    RBT7_BT_CODE_NO : WORD ;
    RBT7_WELD_COUNT : WORD ;
    RBT8_BT_CODE_NO : WORD ;
    RBT8_WELD_COUNT : WORD ;
    RBT9_BT_CODE_NO : WORD ;
    RBT9_WELD_COUNT : WORD ;
    RBT10_BT_CODE_NO : WORD ;
    RBT10_WELD_COUNT : WORD ;
    RBT11_BT_CODE_NO : WORD ;
    RBT11_WELD_COUNT : WORD ;
    RBT12_BT_CODE_NO : WORD ;
    RBT12_WELD_COUNT : WORD ;
    RBT13_BT_CODE_NO : WORD ;
    RBT13_WELD_COUNT : WORD ;
    RBT14_BT_CODE_NO : WORD ;
    RBT14_WELD_COUNT : WORD ;
    RBT15_BT_CODE_NO : WORD ;
    RBT15_WELD_COUNT : WORD ;
    RBT16_BT_CODE_NO : WORD ;
    RBT16_WELD_COUNT : WORD ;
    RBT17_BT_CODE_NO : WORD ;
    RBT17_WELD_COUNT : WORD ;
    RBT18_BT_CODE_NO : WORD ;
    RBT18_WELD_COUNT : WORD ;
    RBT19_BT_CODE_NO : WORD ;
    RBT19_WELD_COUNT : WORD ;
    RBT20_BT_CODE_NO : WORD ;
    RBT20_WELD_COUNT : WORD ;
    RBT21_BT_CODE_NO : WORD ;
    RBT21_WELD_COUNT : WORD ;
    RBT22_BT_CODE_NO : WORD ;
    RBT22_WELD_COUNT : WORD ;
    RBT23_BT_CODE_NO : WORD ;
    RBT23_WELD_COUNT : WORD ;
    RBT24_BT_CODE_NO : WORD ;
    RBT24_WELD_COUNT : WORD ;
    WELD_DETERMINES_RESULT : WORD ;
    WELD_CHECK_SUM : WORD ;
    SPARE1 : WORD ;
   END_STRUCT ;
  END_STRUCT ;
BEGIN
   S702_WELD_BUFF_DATA1.STATION_MAIN := W#16#0;
   S702_WELD_BUFF_DATA1.DISTINCTION_LH_RH := W#16#0;
   S702_WELD_BUFF_DATA1.STAION_NUMBER := W#16#0;
   S702_WELD_BUFF_DATA1.VIN_NUMBER1 := W#16#0;
   S702_WELD_BUFF_DATA1.VIN_NUMBER2 := W#16#0;
   S702_WELD_BUFF_DATA1.VIN_NUMBER3 := W#16#0;
   S702_WELD_BUFF_DATA1.VIN_NUMBER4 := W#16#0;
   S702_WELD_BUFF_DATA1.SEQ_NUMBER1 := W#16#0;
   S702_WELD_BUFF_DATA1.SEQ_NUMBER2 := W#16#0;
   S702_WELD_BUFF_DATA1.RBT1_BT_CODE_NO := W#16#0;
   S702_WELD_BUFF_DATA1.RBT1_WELD_COUNT := W#16#0;
   S702_WELD_BUFF_DATA1.RBT2_BT_CODE_NO := W#16#0;
   S702_WELD_BUFF_DATA1.RBT2_WELD_COUNT := W#16#0;
   S702_WELD_BUFF_DATA1.RBT3_BT_CODE_NO := W#16#0;
   S702_WELD_BUFF_DATA1.RBT3_WELD_COUNT := W#16#0;
   S702_WELD_BUFF_DATA1.RBT4_BT_CODE_NO := W#16#0;
   S702_WELD_BUFF_DATA1.RBT4_WELD_COUNT := W#16#0;
   S702_WELD_BUFF_DATA1.RBT5_BT_CODE_NO := W#16#0;
   S702_WELD_BUFF_DATA1.RBT5_WELD_COUNT := W#16#0;
   S702_WELD_BUFF_DATA1.RBT6_BT_CODE_NO := W#16#0;
   S702_WELD_BUFF_DATA1.RBT6_WELD_COUNT := W#16#0;
   S702_WELD_BUFF_DATA1.RBT7_BT_CODE_NO := W#16#0;
   S702_WELD_BUFF_DATA1.RBT7_WELD_COUNT := W#16#0;
   S702_WELD_BUFF_DATA1.RBT8_BT_CODE_NO := W#16#0;
   S702_WELD_BUFF_DATA1.RBT8_WELD_COUNT := W#16#0;
   S702_WELD_BUFF_DATA1.RBT9_BT_CODE_NO := W#16#0;
   S702_WELD_BUFF_DATA1.RBT9_WELD_COUNT := W#16#0;
   S702_WELD_BUFF_DATA1.RBT10_BT_CODE_NO := W#16#0;
   S702_WELD_BUFF_DATA1.RBT10_WELD_COUNT := W#16#0;
   S702_WELD_BUFF_DATA1.RBT11_BT_CODE_NO := W#16#0;
   S702_WELD_BUFF_DATA1.RBT11_WELD_COUNT := W#16#0;
   S702_WELD_BUFF_DATA1.RBT12_BT_CODE_NO := W#16#0;
   S702_WELD_BUFF_DATA1.RBT12_WELD_COUNT := W#16#0;
   S702_WELD_BUFF_DATA1.RBT13_BT_CODE_NO := W#16#0;
   S702_WELD_BUFF_DATA1.RBT13_WELD_COUNT := W#16#0;
   S702_WELD_BUFF_DATA1.RBT14_BT_CODE_NO := W#16#0;
   S702_WELD_BUFF_DATA1.RBT14_WELD_COUNT := W#16#0;
   S702_WELD_BUFF_DATA1.RBT15_BT_CODE_NO := W#16#0;
   S702_WELD_BUFF_DATA1.RBT15_WELD_COUNT := W#16#0;
   S702_WELD_BUFF_DATA1.RBT16_BT_CODE_NO := W#16#0;
   S702_WELD_BUFF_DATA1.RBT16_WELD_COUNT := W#16#0;
   S702_WELD_BUFF_DATA1.RBT17_BT_CODE_NO := W#16#0;
   S702_WELD_BUFF_DATA1.RBT17_WELD_COUNT := W#16#0;
   S702_WELD_BUFF_DATA1.RBT18_BT_CODE_NO := W#16#0;
   S702_WELD_BUFF_DATA1.RBT18_WELD_COUNT := W#16#0;
   S702_WELD_BUFF_DATA1.RBT19_BT_CODE_NO := W#16#0;
   S702_WELD_BUFF_DATA1.RBT19_WELD_COUNT := W#16#0;
   S702_WELD_BUFF_DATA1.RBT20_BT_CODE_NO := W#16#0;
   S702_WELD_BUFF_DATA1.RBT20_WELD_COUNT := W#16#0;
   S702_WELD_BUFF_DATA1.RBT21_BT_CODE_NO := W#16#0;
   S702_WELD_BUFF_DATA1.RBT21_WELD_COUNT := W#16#0;
   S702_WELD_BUFF_DATA1.RBT22_BT_CODE_NO := W#16#0;
   S702_WELD_BUFF_DATA1.RBT22_WELD_COUNT := W#16#0;
   S702_WELD_BUFF_DATA1.RBT23_BT_CODE_NO := W#16#0;
   S702_WELD_BUFF_DATA1.RBT23_WELD_COUNT := W#16#0;
   S702_WELD_BUFF_DATA1.RBT24_BT_CODE_NO := W#16#0;
   S702_WELD_BUFF_DATA1.RBT24_WELD_COUNT := W#16#0;
   S702_WELD_BUFF_DATA1.WELD_DETERMINES_RESULT := W#16#0;
   S702_WELD_BUFF_DATA1.WELD_CHECK_SUM := W#16#0;
   S702_WELD_BUFF_DATA1.SPARE1 := W#16#0;
   S702_WELD_BUFF_DATA2.STATION_MAIN := W#16#0;
   S702_WELD_BUFF_DATA2.DISTINCTION_LH_RH := W#16#0;
   S702_WELD_BUFF_DATA2.STAION_NUMBER := W#16#0;
   S702_WELD_BUFF_DATA2.VIN_NUMBER1 := W#16#0;
   S702_WELD_BUFF_DATA2.VIN_NUMBER2 := W#16#0;
   S702_WELD_BUFF_DATA2.VIN_NUMBER3 := W#16#0;
   S702_WELD_BUFF_DATA2.VIN_NUMBER4 := W#16#0;
   S702_WELD_BUFF_DATA2.SEQ_NUMBER1 := W#16#0;
   S702_WELD_BUFF_DATA2.SEQ_NUMBER2 := W#16#0;
   S702_WELD_BUFF_DATA2.RBT1_BT_CODE_NO := W#16#0;
   S702_WELD_BUFF_DATA2.RBT1_WELD_COUNT := W#16#0;
   S702_WELD_BUFF_DATA2.RBT2_BT_CODE_NO := W#16#0;
   S702_WELD_BUFF_DATA2.RBT2_WELD_COUNT := W#16#0;
   S702_WELD_BUFF_DATA2.RBT3_BT_CODE_NO := W#16#0;
   S702_WELD_BUFF_DATA2.RBT3_WELD_COUNT := W#16#0;
   S702_WELD_BUFF_DATA2.RBT4_BT_CODE_NO := W#16#0;
   S702_WELD_BUFF_DATA2.RBT4_WELD_COUNT := W#16#0;
   S702_WELD_BUFF_DATA2.RBT5_BT_CODE_NO := W#16#0;
   S702_WELD_BUFF_DATA2.RBT5_WELD_COUNT := W#16#0;
   S702_WELD_BUFF_DATA2.RBT6_BT_CODE_NO := W#16#0;
   S702_WELD_BUFF_DATA2.RBT6_WELD_COUNT := W#16#0;
   S702_WELD_BUFF_DATA2.RBT7_BT_CODE_NO := W#16#0;
   S702_WELD_BUFF_DATA2.RBT7_WELD_COUNT := W#16#0;
   S702_WELD_BUFF_DATA2.RBT8_BT_CODE_NO := W#16#0;
   S702_WELD_BUFF_DATA2.RBT8_WELD_COUNT := W#16#0;
   S702_WELD_BUFF_DATA2.RBT9_BT_CODE_NO := W#16#0;
   S702_WELD_BUFF_DATA2.RBT9_WELD_COUNT := W#16#0;
   S702_WELD_BUFF_DATA2.RBT10_BT_CODE_NO := W#16#0;
   S702_WELD_BUFF_DATA2.RBT10_WELD_COUNT := W#16#0;
   S702_WELD_BUFF_DATA2.RBT11_BT_CODE_NO := W#16#0;
   S702_WELD_BUFF_DATA2.RBT11_WELD_COUNT := W#16#0;
   S702_WELD_BUFF_DATA2.RBT12_BT_CODE_NO := W#16#0;
   S702_WELD_BUFF_DATA2.RBT12_WELD_COUNT := W#16#0;
   S702_WELD_BUFF_DATA2.RBT13_BT_CODE_NO := W#16#0;
   S702_WELD_BUFF_DATA2.RBT13_WELD_COUNT := W#16#0;
   S702_WELD_BUFF_DATA2.RBT14_BT_CODE_NO := W#16#0;
   S702_WELD_BUFF_DATA2.RBT14_WELD_COUNT := W#16#0;
   S702_WELD_BUFF_DATA2.RBT15_BT_CODE_NO := W#16#0;
   S702_WELD_BUFF_DATA2.RBT15_WELD_COUNT := W#16#0;
   S702_WELD_BUFF_DATA2.RBT16_BT_CODE_NO := W#16#0;
   S702_WELD_BUFF_DATA2.RBT16_WELD_COUNT := W#16#0;
   S702_WELD_BUFF_DATA2.RBT17_BT_CODE_NO := W#16#0;
   S702_WELD_BUFF_DATA2.RBT17_WELD_COUNT := W#16#0;
   S702_WELD_BUFF_DATA2.RBT18_BT_CODE_NO := W#16#0;
   S702_WELD_BUFF_DATA2.RBT18_WELD_COUNT := W#16#0;
   S702_WELD_BUFF_DATA2.RBT19_BT_CODE_NO := W#16#0;
   S702_WELD_BUFF_DATA2.RBT19_WELD_COUNT := W#16#0;
   S702_WELD_BUFF_DATA2.RBT20_BT_CODE_NO := W#16#0;
   S702_WELD_BUFF_DATA2.RBT20_WELD_COUNT := W#16#0;
   S702_WELD_BUFF_DATA2.RBT21_BT_CODE_NO := W#16#0;
   S702_WELD_BUFF_DATA2.RBT21_WELD_COUNT := W#16#0;
   S702_WELD_BUFF_DATA2.RBT22_BT_CODE_NO := W#16#0;
   S702_WELD_BUFF_DATA2.RBT22_WELD_COUNT := W#16#0;
   S702_WELD_BUFF_DATA2.RBT23_BT_CODE_NO := W#16#0;
   S702_WELD_BUFF_DATA2.RBT23_WELD_COUNT := W#16#0;
   S702_WELD_BUFF_DATA2.RBT24_BT_CODE_NO := W#16#0;
   S702_WELD_BUFF_DATA2.RBT24_WELD_COUNT := W#16#0;
   S702_WELD_BUFF_DATA2.WELD_DETERMINES_RESULT := W#16#0;
   S702_WELD_BUFF_DATA2.WELD_CHECK_SUM := W#16#0;
   S702_WELD_BUFF_DATA2.SPARE1 := W#16#0;
   S702_WELD_BUFF_DATA3.STATION_MAIN := W#16#0;
   S702_WELD_BUFF_DATA3.DISTINCTION_LH_RH := W#16#0;
   S702_WELD_BUFF_DATA3.STAION_NUMBER := W#16#0;
   S702_WELD_BUFF_DATA3.VIN_NUMBER1 := W#16#0;
   S702_WELD_BUFF_DATA3.VIN_NUMBER2 := W#16#0;
   S702_WELD_BUFF_DATA3.VIN_NUMBER3 := W#16#0;
   S702_WELD_BUFF_DATA3.VIN_NUMBER4 := W#16#0;
   S702_WELD_BUFF_DATA3.SEQ_NUMBER1 := W#16#0;
   S702_WELD_BUFF_DATA3.SEQ_NUMBER2 := W#16#0;
   S702_WELD_BUFF_DATA3.RBT1_BT_CODE_NO := W#16#0;
   S702_WELD_BUFF_DATA3.RBT1_WELD_COUNT := W#16#0;
   S702_WELD_BUFF_DATA3.RBT2_BT_CODE_NO := W#16#0;
   S702_WELD_BUFF_DATA3.RBT2_WELD_COUNT := W#16#0;
   S702_WELD_BUFF_DATA3.RBT3_BT_CODE_NO := W#16#0;
   S702_WELD_BUFF_DATA3.RBT3_WELD_COUNT := W#16#0;
   S702_WELD_BUFF_DATA3.RBT4_BT_CODE_NO := W#16#0;
   S702_WELD_BUFF_DATA3.RBT4_WELD_COUNT := W#16#0;
   S702_WELD_BUFF_DATA3.RBT5_BT_CODE_NO := W#16#0;
   S702_WELD_BUFF_DATA3.RBT5_WELD_COUNT := W#16#0;
   S702_WELD_BUFF_DATA3.RBT6_BT_CODE_NO := W#16#0;
   S702_WELD_BUFF_DATA3.RBT6_WELD_COUNT := W#16#0;
   S702_WELD_BUFF_DATA3.RBT7_BT_CODE_NO := W#16#0;
   S702_WELD_BUFF_DATA3.RBT7_WELD_COUNT := W#16#0;
   S702_WELD_BUFF_DATA3.RBT8_BT_CODE_NO := W#16#0;
   S702_WELD_BUFF_DATA3.RBT8_WELD_COUNT := W#16#0;
   S702_WELD_BUFF_DATA3.RBT9_BT_CODE_NO := W#16#0;
   S702_WELD_BUFF_DATA3.RBT9_WELD_COUNT := W#16#0;
   S702_WELD_BUFF_DATA3.RBT10_BT_CODE_NO := W#16#0;
   S702_WELD_BUFF_DATA3.RBT10_WELD_COUNT := W#16#0;
   S702_WELD_BUFF_DATA3.RBT11_BT_CODE_NO := W#16#0;
   S702_WELD_BUFF_DATA3.RBT11_WELD_COUNT := W#16#0;
   S702_WELD_BUFF_DATA3.RBT12_BT_CODE_NO := W#16#0;
   S702_WELD_BUFF_DATA3.RBT12_WELD_COUNT := W#16#0;
   S702_WELD_BUFF_DATA3.RBT13_BT_CODE_NO := W#16#0;
   S702_WELD_BUFF_DATA3.RBT13_WELD_COUNT := W#16#0;
   S702_WELD_BUFF_DATA3.RBT14_BT_CODE_NO := W#16#0;
   S702_WELD_BUFF_DATA3.RBT14_WELD_COUNT := W#16#0;
   S702_WELD_BUFF_DATA3.RBT15_BT_CODE_NO := W#16#0;
   S702_WELD_BUFF_DATA3.RBT15_WELD_COUNT := W#16#0;
   S702_WELD_BUFF_DATA3.RBT16_BT_CODE_NO := W#16#0;
   S702_WELD_BUFF_DATA3.RBT16_WELD_COUNT := W#16#0;
   S702_WELD_BUFF_DATA3.RBT17_BT_CODE_NO := W#16#0;
   S702_WELD_BUFF_DATA3.RBT17_WELD_COUNT := W#16#0;
   S702_WELD_BUFF_DATA3.RBT18_BT_CODE_NO := W#16#0;
   S702_WELD_BUFF_DATA3.RBT18_WELD_COUNT := W#16#0;
   S702_WELD_BUFF_DATA3.RBT19_BT_CODE_NO := W#16#0;
   S702_WELD_BUFF_DATA3.RBT19_WELD_COUNT := W#16#0;
   S702_WELD_BUFF_DATA3.RBT20_BT_CODE_NO := W#16#0;
   S702_WELD_BUFF_DATA3.RBT20_WELD_COUNT := W#16#0;
   S702_WELD_BUFF_DATA3.RBT21_BT_CODE_NO := W#16#0;
   S702_WELD_BUFF_DATA3.RBT21_WELD_COUNT := W#16#0;
   S702_WELD_BUFF_DATA3.RBT22_BT_CODE_NO := W#16#0;
   S702_WELD_BUFF_DATA3.RBT22_WELD_COUNT := W#16#0;
   S702_WELD_BUFF_DATA3.RBT23_BT_CODE_NO := W#16#0;
   S702_WELD_BUFF_DATA3.RBT23_WELD_COUNT := W#16#0;
   S702_WELD_BUFF_DATA3.RBT24_BT_CODE_NO := W#16#0;
   S702_WELD_BUFF_DATA3.RBT24_WELD_COUNT := W#16#0;
   S702_WELD_BUFF_DATA3.WELD_DETERMINES_RESULT := W#16#0;
   S702_WELD_BUFF_DATA3.WELD_CHECK_SUM := W#16#0;
   S702_WELD_BUFF_DATA3.SPARE1 := W#16#0;
   S702_WELD_BUFF_DATA4.STATION_MAIN := W#16#0;
   S702_WELD_BUFF_DATA4.DISTINCTION_LH_RH := W#16#0;
   S702_WELD_BUFF_DATA4.STAION_NUMBER := W#16#0;
   S702_WELD_BUFF_DATA4.VIN_NUMBER1 := W#16#0;
   S702_WELD_BUFF_DATA4.VIN_NUMBER2 := W#16#0;
   S702_WELD_BUFF_DATA4.VIN_NUMBER3 := W#16#0;
   S702_WELD_BUFF_DATA4.VIN_NUMBER4 := W#16#0;
   S702_WELD_BUFF_DATA4.SEQ_NUMBER1 := W#16#0;
   S702_WELD_BUFF_DATA4.SEQ_NUMBER2 := W#16#0;
   S702_WELD_BUFF_DATA4.RBT1_BT_CODE_NO := W#16#0;
   S702_WELD_BUFF_DATA4.RBT1_WELD_COUNT := W#16#0;
   S702_WELD_BUFF_DATA4.RBT2_BT_CODE_NO := W#16#0;
   S702_WELD_BUFF_DATA4.RBT2_WELD_COUNT := W#16#0;
   S702_WELD_BUFF_DATA4.RBT3_BT_CODE_NO := W#16#0;
   S702_WELD_BUFF_DATA4.RBT3_WELD_COUNT := W#16#0;
   S702_WELD_BUFF_DATA4.RBT4_BT_CODE_NO := W#16#0;
   S702_WELD_BUFF_DATA4.RBT4_WELD_COUNT := W#16#0;
   S702_WELD_BUFF_DATA4.RBT5_BT_CODE_NO := W#16#0;
   S702_WELD_BUFF_DATA4.RBT5_WELD_COUNT := W#16#0;
   S702_WELD_BUFF_DATA4.RBT6_BT_CODE_NO := W#16#0;
   S702_WELD_BUFF_DATA4.RBT6_WELD_COUNT := W#16#0;
   S702_WELD_BUFF_DATA4.RBT7_BT_CODE_NO := W#16#0;
   S702_WELD_BUFF_DATA4.RBT7_WELD_COUNT := W#16#0;
   S702_WELD_BUFF_DATA4.RBT8_BT_CODE_NO := W#16#0;
   S702_WELD_BUFF_DATA4.RBT8_WELD_COUNT := W#16#0;
   S702_WELD_BUFF_DATA4.RBT9_BT_CODE_NO := W#16#0;
   S702_WELD_BUFF_DATA4.RBT9_WELD_COUNT := W#16#0;
   S702_WELD_BUFF_DATA4.RBT10_BT_CODE_NO := W#16#0;
   S702_WELD_BUFF_DATA4.RBT10_WELD_COUNT := W#16#0;
   S702_WELD_BUFF_DATA4.RBT11_BT_CODE_NO := W#16#0;
   S702_WELD_BUFF_DATA4.RBT11_WELD_COUNT := W#16#0;
   S702_WELD_BUFF_DATA4.RBT12_BT_CODE_NO := W#16#0;
   S702_WELD_BUFF_DATA4.RBT12_WELD_COUNT := W#16#0;
   S702_WELD_BUFF_DATA4.RBT13_BT_CODE_NO := W#16#0;
   S702_WELD_BUFF_DATA4.RBT13_WELD_COUNT := W#16#0;
   S702_WELD_BUFF_DATA4.RBT14_BT_CODE_NO := W#16#0;
   S702_WELD_BUFF_DATA4.RBT14_WELD_COUNT := W#16#0;
   S702_WELD_BUFF_DATA4.RBT15_BT_CODE_NO := W#16#0;
   S702_WELD_BUFF_DATA4.RBT15_WELD_COUNT := W#16#0;
   S702_WELD_BUFF_DATA4.RBT16_BT_CODE_NO := W#16#0;
   S702_WELD_BUFF_DATA4.RBT16_WELD_COUNT := W#16#0;
   S702_WELD_BUFF_DATA4.RBT17_BT_CODE_NO := W#16#0;
   S702_WELD_BUFF_DATA4.RBT17_WELD_COUNT := W#16#0;
   S702_WELD_BUFF_DATA4.RBT18_BT_CODE_NO := W#16#0;
   S702_WELD_BUFF_DATA4.RBT18_WELD_COUNT := W#16#0;
   S702_WELD_BUFF_DATA4.RBT19_BT_CODE_NO := W#16#0;
   S702_WELD_BUFF_DATA4.RBT19_WELD_COUNT := W#16#0;
   S702_WELD_BUFF_DATA4.RBT20_BT_CODE_NO := W#16#0;
   S702_WELD_BUFF_DATA4.RBT20_WELD_COUNT := W#16#0;
   S702_WELD_BUFF_DATA4.RBT21_BT_CODE_NO := W#16#0;
   S702_WELD_BUFF_DATA4.RBT21_WELD_COUNT := W#16#0;
   S702_WELD_BUFF_DATA4.RBT22_BT_CODE_NO := W#16#0;
   S702_WELD_BUFF_DATA4.RBT22_WELD_COUNT := W#16#0;
   S702_WELD_BUFF_DATA4.RBT23_BT_CODE_NO := W#16#0;
   S702_WELD_BUFF_DATA4.RBT23_WELD_COUNT := W#16#0;
   S702_WELD_BUFF_DATA4.RBT24_BT_CODE_NO := W#16#0;
   S702_WELD_BUFF_DATA4.RBT24_WELD_COUNT := W#16#0;
   S702_WELD_BUFF_DATA4.WELD_DETERMINES_RESULT := W#16#0;
   S702_WELD_BUFF_DATA4.WELD_CHECK_SUM := W#16#0;
   S702_WELD_BUFF_DATA4.SPARE1 := W#16#0;
   S702_WELD_BUFF_DATA5.STATION_MAIN := W#16#0;
   S702_WELD_BUFF_DATA5.DISTINCTION_LH_RH := W#16#0;
   S702_WELD_BUFF_DATA5.STAION_NUMBER := W#16#0;
   S702_WELD_BUFF_DATA5.VIN_NUMBER1 := W#16#0;
   S702_WELD_BUFF_DATA5.VIN_NUMBER2 := W#16#0;
   S702_WELD_BUFF_DATA5.VIN_NUMBER3 := W#16#0;
   S702_WELD_BUFF_DATA5.VIN_NUMBER4 := W#16#0;
   S702_WELD_BUFF_DATA5.SEQ_NUMBER1 := W#16#0;
   S702_WELD_BUFF_DATA5.SEQ_NUMBER2 := W#16#0;
   S702_WELD_BUFF_DATA5.RBT1_BT_CODE_NO := W#16#0;
   S702_WELD_BUFF_DATA5.RBT1_WELD_COUNT := W#16#0;
   S702_WELD_BUFF_DATA5.RBT2_BT_CODE_NO := W#16#0;
   S702_WELD_BUFF_DATA5.RBT2_WELD_COUNT := W#16#0;
   S702_WELD_BUFF_DATA5.RBT3_BT_CODE_NO := W#16#0;
   S702_WELD_BUFF_DATA5.RBT3_WELD_COUNT := W#16#0;
   S702_WELD_BUFF_DATA5.RBT4_BT_CODE_NO := W#16#0;
   S702_WELD_BUFF_DATA5.RBT4_WELD_COUNT := W#16#0;
   S702_WELD_BUFF_DATA5.RBT5_BT_CODE_NO := W#16#0;
   S702_WELD_BUFF_DATA5.RBT5_WELD_COUNT := W#16#0;
   S702_WELD_BUFF_DATA5.RBT6_BT_CODE_NO := W#16#0;
   S702_WELD_BUFF_DATA5.RBT6_WELD_COUNT := W#16#0;
   S702_WELD_BUFF_DATA5.RBT7_BT_CODE_NO := W#16#0;
   S702_WELD_BUFF_DATA5.RBT7_WELD_COUNT := W#16#0;
   S702_WELD_BUFF_DATA5.RBT8_BT_CODE_NO := W#16#0;
   S702_WELD_BUFF_DATA5.RBT8_WELD_COUNT := W#16#0;
   S702_WELD_BUFF_DATA5.RBT9_BT_CODE_NO := W#16#0;
   S702_WELD_BUFF_DATA5.RBT9_WELD_COUNT := W#16#0;
   S702_WELD_BUFF_DATA5.RBT10_BT_CODE_NO := W#16#0;
   S702_WELD_BUFF_DATA5.RBT10_WELD_COUNT := W#16#0;
   S702_WELD_BUFF_DATA5.RBT11_BT_CODE_NO := W#16#0;
   S702_WELD_BUFF_DATA5.RBT11_WELD_COUNT := W#16#0;
   S702_WELD_BUFF_DATA5.RBT12_BT_CODE_NO := W#16#0;
   S702_WELD_BUFF_DATA5.RBT12_WELD_COUNT := W#16#0;
   S702_WELD_BUFF_DATA5.RBT13_BT_CODE_NO := W#16#0;
   S702_WELD_BUFF_DATA5.RBT13_WELD_COUNT := W#16#0;
   S702_WELD_BUFF_DATA5.RBT14_BT_CODE_NO := W#16#0;
   S702_WELD_BUFF_DATA5.RBT14_WELD_COUNT := W#16#0;
   S702_WELD_BUFF_DATA5.RBT15_BT_CODE_NO := W#16#0;
   S702_WELD_BUFF_DATA5.RBT15_WELD_COUNT := W#16#0;
   S702_WELD_BUFF_DATA5.RBT16_BT_CODE_NO := W#16#0;
   S702_WELD_BUFF_DATA5.RBT16_WELD_COUNT := W#16#0;
   S702_WELD_BUFF_DATA5.RBT17_BT_CODE_NO := W#16#0;
   S702_WELD_BUFF_DATA5.RBT17_WELD_COUNT := W#16#0;
   S702_WELD_BUFF_DATA5.RBT18_BT_CODE_NO := W#16#0;
   S702_WELD_BUFF_DATA5.RBT18_WELD_COUNT := W#16#0;
   S702_WELD_BUFF_DATA5.RBT19_BT_CODE_NO := W#16#0;
   S702_WELD_BUFF_DATA5.RBT19_WELD_COUNT := W#16#0;
   S702_WELD_BUFF_DATA5.RBT20_BT_CODE_NO := W#16#0;
   S702_WELD_BUFF_DATA5.RBT20_WELD_COUNT := W#16#0;
   S702_WELD_BUFF_DATA5.RBT21_BT_CODE_NO := W#16#0;
   S702_WELD_BUFF_DATA5.RBT21_WELD_COUNT := W#16#0;
   S702_WELD_BUFF_DATA5.RBT22_BT_CODE_NO := W#16#0;
   S702_WELD_BUFF_DATA5.RBT22_WELD_COUNT := W#16#0;
   S702_WELD_BUFF_DATA5.RBT23_BT_CODE_NO := W#16#0;
   S702_WELD_BUFF_DATA5.RBT23_WELD_COUNT := W#16#0;
   S702_WELD_BUFF_DATA5.RBT24_BT_CODE_NO := W#16#0;
   S702_WELD_BUFF_DATA5.RBT24_WELD_COUNT := W#16#0;
   S702_WELD_BUFF_DATA5.WELD_DETERMINES_RESULT := W#16#0;
   S702_WELD_BUFF_DATA5.WELD_CHECK_SUM := W#16#0;
   S702_WELD_BUFF_DATA5.SPARE1 := W#16#0;
   S702_WELD_BUFF_DATA6.STATION_MAIN := W#16#0;
   S702_WELD_BUFF_DATA6.DISTINCTION_LH_RH := W#16#0;
   S702_WELD_BUFF_DATA6.STAION_NUMBER := W#16#0;
   S702_WELD_BUFF_DATA6.VIN_NUMBER1 := W#16#0;
   S702_WELD_BUFF_DATA6.VIN_NUMBER2 := W#16#0;
   S702_WELD_BUFF_DATA6.VIN_NUMBER3 := W#16#0;
   S702_WELD_BUFF_DATA6.VIN_NUMBER4 := W#16#0;
   S702_WELD_BUFF_DATA6.SEQ_NUMBER1 := W#16#0;
   S702_WELD_BUFF_DATA6.SEQ_NUMBER2 := W#16#0;
   S702_WELD_BUFF_DATA6.RBT1_BT_CODE_NO := W#16#0;
   S702_WELD_BUFF_DATA6.RBT1_WELD_COUNT := W#16#0;
   S702_WELD_BUFF_DATA6.RBT2_BT_CODE_NO := W#16#0;
   S702_WELD_BUFF_DATA6.RBT2_WELD_COUNT := W#16#0;
   S702_WELD_BUFF_DATA6.RBT3_BT_CODE_NO := W#16#0;
   S702_WELD_BUFF_DATA6.RBT3_WELD_COUNT := W#16#0;
   S702_WELD_BUFF_DATA6.RBT4_BT_CODE_NO := W#16#0;
   S702_WELD_BUFF_DATA6.RBT4_WELD_COUNT := W#16#0;
   S702_WELD_BUFF_DATA6.RBT5_BT_CODE_NO := W#16#0;
   S702_WELD_BUFF_DATA6.RBT5_WELD_COUNT := W#16#0;
   S702_WELD_BUFF_DATA6.RBT6_BT_CODE_NO := W#16#0;
   S702_WELD_BUFF_DATA6.RBT6_WELD_COUNT := W#16#0;
   S702_WELD_BUFF_DATA6.RBT7_BT_CODE_NO := W#16#0;
   S702_WELD_BUFF_DATA6.RBT7_WELD_COUNT := W#16#0;
   S702_WELD_BUFF_DATA6.RBT8_BT_CODE_NO := W#16#0;
   S702_WELD_BUFF_DATA6.RBT8_WELD_COUNT := W#16#0;
   S702_WELD_BUFF_DATA6.RBT9_BT_CODE_NO := W#16#0;
   S702_WELD_BUFF_DATA6.RBT9_WELD_COUNT := W#16#0;
   S702_WELD_BUFF_DATA6.RBT10_BT_CODE_NO := W#16#0;
   S702_WELD_BUFF_DATA6.RBT10_WELD_COUNT := W#16#0;
   S702_WELD_BUFF_DATA6.RBT11_BT_CODE_NO := W#16#0;
   S702_WELD_BUFF_DATA6.RBT11_WELD_COUNT := W#16#0;
   S702_WELD_BUFF_DATA6.RBT12_BT_CODE_NO := W#16#0;
   S702_WELD_BUFF_DATA6.RBT12_WELD_COUNT := W#16#0;
   S702_WELD_BUFF_DATA6.RBT13_BT_CODE_NO := W#16#0;
   S702_WELD_BUFF_DATA6.RBT13_WELD_COUNT := W#16#0;
   S702_WELD_BUFF_DATA6.RBT14_BT_CODE_NO := W#16#0;
   S702_WELD_BUFF_DATA6.RBT14_WELD_COUNT := W#16#0;
   S702_WELD_BUFF_DATA6.RBT15_BT_CODE_NO := W#16#0;
   S702_WELD_BUFF_DATA6.RBT15_WELD_COUNT := W#16#0;
   S702_WELD_BUFF_DATA6.RBT16_BT_CODE_NO := W#16#0;
   S702_WELD_BUFF_DATA6.RBT16_WELD_COUNT := W#16#0;
   S702_WELD_BUFF_DATA6.RBT17_BT_CODE_NO := W#16#0;
   S702_WELD_BUFF_DATA6.RBT17_WELD_COUNT := W#16#0;
   S702_WELD_BUFF_DATA6.RBT18_BT_CODE_NO := W#16#0;
   S702_WELD_BUFF_DATA6.RBT18_WELD_COUNT := W#16#0;
   S702_WELD_BUFF_DATA6.RBT19_BT_CODE_NO := W#16#0;
   S702_WELD_BUFF_DATA6.RBT19_WELD_COUNT := W#16#0;
   S702_WELD_BUFF_DATA6.RBT20_BT_CODE_NO := W#16#0;
   S702_WELD_BUFF_DATA6.RBT20_WELD_COUNT := W#16#0;
   S702_WELD_BUFF_DATA6.RBT21_BT_CODE_NO := W#16#0;
   S702_WELD_BUFF_DATA6.RBT21_WELD_COUNT := W#16#0;
   S702_WELD_BUFF_DATA6.RBT22_BT_CODE_NO := W#16#0;
   S702_WELD_BUFF_DATA6.RBT22_WELD_COUNT := W#16#0;
   S702_WELD_BUFF_DATA6.RBT23_BT_CODE_NO := W#16#0;
   S702_WELD_BUFF_DATA6.RBT23_WELD_COUNT := W#16#0;
   S702_WELD_BUFF_DATA6.RBT24_BT_CODE_NO := W#16#0;
   S702_WELD_BUFF_DATA6.RBT24_WELD_COUNT := W#16#0;
   S702_WELD_BUFF_DATA6.WELD_DETERMINES_RESULT := W#16#0;
   S702_WELD_BUFF_DATA6.WELD_CHECK_SUM := W#16#0;
   S702_WELD_BUFF_DATA6.SPARE1 := W#16#0;
   S702_WELD_BUFF_DATA7.STATION_MAIN := W#16#0;
   S702_WELD_BUFF_DATA7.DISTINCTION_LH_RH := W#16#0;
   S702_WELD_BUFF_DATA7.STAION_NUMBER := W#16#0;
   S702_WELD_BUFF_DATA7.VIN_NUMBER1 := W#16#0;
   S702_WELD_BUFF_DATA7.VIN_NUMBER2 := W#16#0;
   S702_WELD_BUFF_DATA7.VIN_NUMBER3 := W#16#0;
   S702_WELD_BUFF_DATA7.VIN_NUMBER4 := W#16#0;
   S702_WELD_BUFF_DATA7.SEQ_NUMBER1 := W#16#0;
   S702_WELD_BUFF_DATA7.SEQ_NUMBER2 := W#16#0;
   S702_WELD_BUFF_DATA7.RBT1_BT_CODE_NO := W#16#0;
   S702_WELD_BUFF_DATA7.RBT1_WELD_COUNT := W#16#0;
   S702_WELD_BUFF_DATA7.RBT2_BT_CODE_NO := W#16#0;
   S702_WELD_BUFF_DATA7.RBT2_WELD_COUNT := W#16#0;
   S702_WELD_BUFF_DATA7.RBT3_BT_CODE_NO := W#16#0;
   S702_WELD_BUFF_DATA7.RBT3_WELD_COUNT := W#16#0;
   S702_WELD_BUFF_DATA7.RBT4_BT_CODE_NO := W#16#0;
   S702_WELD_BUFF_DATA7.RBT4_WELD_COUNT := W#16#0;
   S702_WELD_BUFF_DATA7.RBT5_BT_CODE_NO := W#16#0;
   S702_WELD_BUFF_DATA7.RBT5_WELD_COUNT := W#16#0;
   S702_WELD_BUFF_DATA7.RBT6_BT_CODE_NO := W#16#0;
   S702_WELD_BUFF_DATA7.RBT6_WELD_COUNT := W#16#0;
   S702_WELD_BUFF_DATA7.RBT7_BT_CODE_NO := W#16#0;
   S702_WELD_BUFF_DATA7.RBT7_WELD_COUNT := W#16#0;
   S702_WELD_BUFF_DATA7.RBT8_BT_CODE_NO := W#16#0;
   S702_WELD_BUFF_DATA7.RBT8_WELD_COUNT := W#16#0;
   S702_WELD_BUFF_DATA7.RBT9_BT_CODE_NO := W#16#0;
   S702_WELD_BUFF_DATA7.RBT9_WELD_COUNT := W#16#0;
   S702_WELD_BUFF_DATA7.RBT10_BT_CODE_NO := W#16#0;
   S702_WELD_BUFF_DATA7.RBT10_WELD_COUNT := W#16#0;
   S702_WELD_BUFF_DATA7.RBT11_BT_CODE_NO := W#16#0;
   S702_WELD_BUFF_DATA7.RBT11_WELD_COUNT := W#16#0;
   S702_WELD_BUFF_DATA7.RBT12_BT_CODE_NO := W#16#0;
   S702_WELD_BUFF_DATA7.RBT12_WELD_COUNT := W#16#0;
   S702_WELD_BUFF_DATA7.RBT13_BT_CODE_NO := W#16#0;
   S702_WELD_BUFF_DATA7.RBT13_WELD_COUNT := W#16#0;
   S702_WELD_BUFF_DATA7.RBT14_BT_CODE_NO := W#16#0;
   S702_WELD_BUFF_DATA7.RBT14_WELD_COUNT := W#16#0;
   S702_WELD_BUFF_DATA7.RBT15_BT_CODE_NO := W#16#0;
   S702_WELD_BUFF_DATA7.RBT15_WELD_COUNT := W#16#0;
   S702_WELD_BUFF_DATA7.RBT16_BT_CODE_NO := W#16#0;
   S702_WELD_BUFF_DATA7.RBT16_WELD_COUNT := W#16#0;
   S702_WELD_BUFF_DATA7.RBT17_BT_CODE_NO := W#16#0;
   S702_WELD_BUFF_DATA7.RBT17_WELD_COUNT := W#16#0;
   S702_WELD_BUFF_DATA7.RBT18_BT_CODE_NO := W#16#0;
   S702_WELD_BUFF_DATA7.RBT18_WELD_COUNT := W#16#0;
   S702_WELD_BUFF_DATA7.RBT19_BT_CODE_NO := W#16#0;
   S702_WELD_BUFF_DATA7.RBT19_WELD_COUNT := W#16#0;
   S702_WELD_BUFF_DATA7.RBT20_BT_CODE_NO := W#16#0;
   S702_WELD_BUFF_DATA7.RBT20_WELD_COUNT := W#16#0;
   S702_WELD_BUFF_DATA7.RBT21_BT_CODE_NO := W#16#0;
   S702_WELD_BUFF_DATA7.RBT21_WELD_COUNT := W#16#0;
   S702_WELD_BUFF_DATA7.RBT22_BT_CODE_NO := W#16#0;
   S702_WELD_BUFF_DATA7.RBT22_WELD_COUNT := W#16#0;
   S702_WELD_BUFF_DATA7.RBT23_BT_CODE_NO := W#16#0;
   S702_WELD_BUFF_DATA7.RBT23_WELD_COUNT := W#16#0;
   S702_WELD_BUFF_DATA7.RBT24_BT_CODE_NO := W#16#0;
   S702_WELD_BUFF_DATA7.RBT24_WELD_COUNT := W#16#0;
   S702_WELD_BUFF_DATA7.WELD_DETERMINES_RESULT := W#16#0;
   S702_WELD_BUFF_DATA7.WELD_CHECK_SUM := W#16#0;
   S702_WELD_BUFF_DATA7.SPARE1 := W#16#0;
   S702_WELD_BUFF_DATA8.STATION_MAIN := W#16#0;
   S702_WELD_BUFF_DATA8.DISTINCTION_LH_RH := W#16#0;
   S702_WELD_BUFF_DATA8.STAION_NUMBER := W#16#0;
   S702_WELD_BUFF_DATA8.VIN_NUMBER1 := W#16#0;
   S702_WELD_BUFF_DATA8.VIN_NUMBER2 := W#16#0;
   S702_WELD_BUFF_DATA8.VIN_NUMBER3 := W#16#0;
   S702_WELD_BUFF_DATA8.VIN_NUMBER4 := W#16#0;
   S702_WELD_BUFF_DATA8.SEQ_NUMBER1 := W#16#0;
   S702_WELD_BUFF_DATA8.SEQ_NUMBER2 := W#16#0;
   S702_WELD_BUFF_DATA8.RBT1_BT_CODE_NO := W#16#0;
   S702_WELD_BUFF_DATA8.RBT1_WELD_COUNT := W#16#0;
   S702_WELD_BUFF_DATA8.RBT2_BT_CODE_NO := W#16#0;
   S702_WELD_BUFF_DATA8.RBT2_WELD_COUNT := W#16#0;
   S702_WELD_BUFF_DATA8.RBT3_BT_CODE_NO := W#16#0;
   S702_WELD_BUFF_DATA8.RBT3_WELD_COUNT := W#16#0;
   S702_WELD_BUFF_DATA8.RBT4_BT_CODE_NO := W#16#0;
   S702_WELD_BUFF_DATA8.RBT4_WELD_COUNT := W#16#0;
   S702_WELD_BUFF_DATA8.RBT5_BT_CODE_NO := W#16#0;
   S702_WELD_BUFF_DATA8.RBT5_WELD_COUNT := W#16#0;
   S702_WELD_BUFF_DATA8.RBT6_BT_CODE_NO := W#16#0;
   S702_WELD_BUFF_DATA8.RBT6_WELD_COUNT := W#16#0;
   S702_WELD_BUFF_DATA8.RBT7_BT_CODE_NO := W#16#0;
   S702_WELD_BUFF_DATA8.RBT7_WELD_COUNT := W#16#0;
   S702_WELD_BUFF_DATA8.RBT8_BT_CODE_NO := W#16#0;
   S702_WELD_BUFF_DATA8.RBT8_WELD_COUNT := W#16#0;
   S702_WELD_BUFF_DATA8.RBT9_BT_CODE_NO := W#16#0;
   S702_WELD_BUFF_DATA8.RBT9_WELD_COUNT := W#16#0;
   S702_WELD_BUFF_DATA8.RBT10_BT_CODE_NO := W#16#0;
   S702_WELD_BUFF_DATA8.RBT10_WELD_COUNT := W#16#0;
   S702_WELD_BUFF_DATA8.RBT11_BT_CODE_NO := W#16#0;
   S702_WELD_BUFF_DATA8.RBT11_WELD_COUNT := W#16#0;
   S702_WELD_BUFF_DATA8.RBT12_BT_CODE_NO := W#16#0;
   S702_WELD_BUFF_DATA8.RBT12_WELD_COUNT := W#16#0;
   S702_WELD_BUFF_DATA8.RBT13_BT_CODE_NO := W#16#0;
   S702_WELD_BUFF_DATA8.RBT13_WELD_COUNT := W#16#0;
   S702_WELD_BUFF_DATA8.RBT14_BT_CODE_NO := W#16#0;
   S702_WELD_BUFF_DATA8.RBT14_WELD_COUNT := W#16#0;
   S702_WELD_BUFF_DATA8.RBT15_BT_CODE_NO := W#16#0;
   S702_WELD_BUFF_DATA8.RBT15_WELD_COUNT := W#16#0;
   S702_WELD_BUFF_DATA8.RBT16_BT_CODE_NO := W#16#0;
   S702_WELD_BUFF_DATA8.RBT16_WELD_COUNT := W#16#0;
   S702_WELD_BUFF_DATA8.RBT17_BT_CODE_NO := W#16#0;
   S702_WELD_BUFF_DATA8.RBT17_WELD_COUNT := W#16#0;
   S702_WELD_BUFF_DATA8.RBT18_BT_CODE_NO := W#16#0;
   S702_WELD_BUFF_DATA8.RBT18_WELD_COUNT := W#16#0;
   S702_WELD_BUFF_DATA8.RBT19_BT_CODE_NO := W#16#0;
   S702_WELD_BUFF_DATA8.RBT19_WELD_COUNT := W#16#0;
   S702_WELD_BUFF_DATA8.RBT20_BT_CODE_NO := W#16#0;
   S702_WELD_BUFF_DATA8.RBT20_WELD_COUNT := W#16#0;
   S702_WELD_BUFF_DATA8.RBT21_BT_CODE_NO := W#16#0;
   S702_WELD_BUFF_DATA8.RBT21_WELD_COUNT := W#16#0;
   S702_WELD_BUFF_DATA8.RBT22_BT_CODE_NO := W#16#0;
   S702_WELD_BUFF_DATA8.RBT22_WELD_COUNT := W#16#0;
   S702_WELD_BUFF_DATA8.RBT23_BT_CODE_NO := W#16#0;
   S702_WELD_BUFF_DATA8.RBT23_WELD_COUNT := W#16#0;
   S702_WELD_BUFF_DATA8.RBT24_BT_CODE_NO := W#16#0;
   S702_WELD_BUFF_DATA8.RBT24_WELD_COUNT := W#16#0;
   S702_WELD_BUFF_DATA8.WELD_DETERMINES_RESULT := W#16#0;
   S702_WELD_BUFF_DATA8.WELD_CHECK_SUM := W#16#0;
   S702_WELD_BUFF_DATA8.SPARE1 := W#16#0;
   S702_WELD_BUFF_DATA9.STATION_MAIN := W#16#0;
   S702_WELD_BUFF_DATA9.DISTINCTION_LH_RH := W#16#0;
   S702_WELD_BUFF_DATA9.STAION_NUMBER := W#16#0;
   S702_WELD_BUFF_DATA9.VIN_NUMBER1 := W#16#0;
   S702_WELD_BUFF_DATA9.VIN_NUMBER2 := W#16#0;
   S702_WELD_BUFF_DATA9.VIN_NUMBER3 := W#16#0;
   S702_WELD_BUFF_DATA9.VIN_NUMBER4 := W#16#0;
   S702_WELD_BUFF_DATA9.SEQ_NUMBER1 := W#16#0;
   S702_WELD_BUFF_DATA9.SEQ_NUMBER2 := W#16#0;
   S702_WELD_BUFF_DATA9.RBT1_BT_CODE_NO := W#16#0;
   S702_WELD_BUFF_DATA9.RBT1_WELD_COUNT := W#16#0;
   S702_WELD_BUFF_DATA9.RBT2_BT_CODE_NO := W#16#0;
   S702_WELD_BUFF_DATA9.RBT2_WELD_COUNT := W#16#0;
   S702_WELD_BUFF_DATA9.RBT3_BT_CODE_NO := W#16#0;
   S702_WELD_BUFF_DATA9.RBT3_WELD_COUNT := W#16#0;
   S702_WELD_BUFF_DATA9.RBT4_BT_CODE_NO := W#16#0;
   S702_WELD_BUFF_DATA9.RBT4_WELD_COUNT := W#16#0;
   S702_WELD_BUFF_DATA9.RBT5_BT_CODE_NO := W#16#0;
   S702_WELD_BUFF_DATA9.RBT5_WELD_COUNT := W#16#0;
   S702_WELD_BUFF_DATA9.RBT6_BT_CODE_NO := W#16#0;
   S702_WELD_BUFF_DATA9.RBT6_WELD_COUNT := W#16#0;
   S702_WELD_BUFF_DATA9.RBT7_BT_CODE_NO := W#16#0;
   S702_WELD_BUFF_DATA9.RBT7_WELD_COUNT := W#16#0;
   S702_WELD_BUFF_DATA9.RBT8_BT_CODE_NO := W#16#0;
   S702_WELD_BUFF_DATA9.RBT8_WELD_COUNT := W#16#0;
   S702_WELD_BUFF_DATA9.RBT9_BT_CODE_NO := W#16#0;
   S702_WELD_BUFF_DATA9.RBT9_WELD_COUNT := W#16#0;
   S702_WELD_BUFF_DATA9.RBT10_BT_CODE_NO := W#16#0;
   S702_WELD_BUFF_DATA9.RBT10_WELD_COUNT := W#16#0;
   S702_WELD_BUFF_DATA9.RBT11_BT_CODE_NO := W#16#0;
   S702_WELD_BUFF_DATA9.RBT11_WELD_COUNT := W#16#0;
   S702_WELD_BUFF_DATA9.RBT12_BT_CODE_NO := W#16#0;
   S702_WELD_BUFF_DATA9.RBT12_WELD_COUNT := W#16#0;
   S702_WELD_BUFF_DATA9.RBT13_BT_CODE_NO := W#16#0;
   S702_WELD_BUFF_DATA9.RBT13_WELD_COUNT := W#16#0;
   S702_WELD_BUFF_DATA9.RBT14_BT_CODE_NO := W#16#0;
   S702_WELD_BUFF_DATA9.RBT14_WELD_COUNT := W#16#0;
   S702_WELD_BUFF_DATA9.RBT15_BT_CODE_NO := W#16#0;
   S702_WELD_BUFF_DATA9.RBT15_WELD_COUNT := W#16#0;
   S702_WELD_BUFF_DATA9.RBT16_BT_CODE_NO := W#16#0;
   S702_WELD_BUFF_DATA9.RBT16_WELD_COUNT := W#16#0;
   S702_WELD_BUFF_DATA9.RBT17_BT_CODE_NO := W#16#0;
   S702_WELD_BUFF_DATA9.RBT17_WELD_COUNT := W#16#0;
   S702_WELD_BUFF_DATA9.RBT18_BT_CODE_NO := W#16#0;
   S702_WELD_BUFF_DATA9.RBT18_WELD_COUNT := W#16#0;
   S702_WELD_BUFF_DATA9.RBT19_BT_CODE_NO := W#16#0;
   S702_WELD_BUFF_DATA9.RBT19_WELD_COUNT := W#16#0;
   S702_WELD_BUFF_DATA9.RBT20_BT_CODE_NO := W#16#0;
   S702_WELD_BUFF_DATA9.RBT20_WELD_COUNT := W#16#0;
   S702_WELD_BUFF_DATA9.RBT21_BT_CODE_NO := W#16#0;
   S702_WELD_BUFF_DATA9.RBT21_WELD_COUNT := W#16#0;
   S702_WELD_BUFF_DATA9.RBT22_BT_CODE_NO := W#16#0;
   S702_WELD_BUFF_DATA9.RBT22_WELD_COUNT := W#16#0;
   S702_WELD_BUFF_DATA9.RBT23_BT_CODE_NO := W#16#0;
   S702_WELD_BUFF_DATA9.RBT23_WELD_COUNT := W#16#0;
   S702_WELD_BUFF_DATA9.RBT24_BT_CODE_NO := W#16#0;
   S702_WELD_BUFF_DATA9.RBT24_WELD_COUNT := W#16#0;
   S702_WELD_BUFF_DATA9.WELD_DETERMINES_RESULT := W#16#0;
   S702_WELD_BUFF_DATA9.WELD_CHECK_SUM := W#16#0;
   S702_WELD_BUFF_DATA9.SPARE1 := W#16#0;
   S702_WELD_BUFF_DATA10.STATION_MAIN := W#16#0;
   S702_WELD_BUFF_DATA10.DISTINCTION_LH_RH := W#16#0;
   S702_WELD_BUFF_DATA10.STAION_NUMBER := W#16#0;
   S702_WELD_BUFF_DATA10.VIN_NUMBER1 := W#16#0;
   S702_WELD_BUFF_DATA10.VIN_NUMBER2 := W#16#0;
   S702_WELD_BUFF_DATA10.VIN_NUMBER3 := W#16#0;
   S702_WELD_BUFF_DATA10.VIN_NUMBER4 := W#16#0;
   S702_WELD_BUFF_DATA10.SEQ_NUMBER1 := W#16#0;
   S702_WELD_BUFF_DATA10.SEQ_NUMBER2 := W#16#0;
   S702_WELD_BUFF_DATA10.RBT1_BT_CODE_NO := W#16#0;
   S702_WELD_BUFF_DATA10.RBT1_WELD_COUNT := W#16#0;
   S702_WELD_BUFF_DATA10.RBT2_BT_CODE_NO := W#16#0;
   S702_WELD_BUFF_DATA10.RBT2_WELD_COUNT := W#16#0;
   S702_WELD_BUFF_DATA10.RBT3_BT_CODE_NO := W#16#0;
   S702_WELD_BUFF_DATA10.RBT3_WELD_COUNT := W#16#0;
   S702_WELD_BUFF_DATA10.RBT4_BT_CODE_NO := W#16#0;
   S702_WELD_BUFF_DATA10.RBT4_WELD_COUNT := W#16#0;
   S702_WELD_BUFF_DATA10.RBT5_BT_CODE_NO := W#16#0;
   S702_WELD_BUFF_DATA10.RBT5_WELD_COUNT := W#16#0;
   S702_WELD_BUFF_DATA10.RBT6_BT_CODE_NO := W#16#0;
   S702_WELD_BUFF_DATA10.RBT6_WELD_COUNT := W#16#0;
   S702_WELD_BUFF_DATA10.RBT7_BT_CODE_NO := W#16#0;
   S702_WELD_BUFF_DATA10.RBT7_WELD_COUNT := W#16#0;
   S702_WELD_BUFF_DATA10.RBT8_BT_CODE_NO := W#16#0;
   S702_WELD_BUFF_DATA10.RBT8_WELD_COUNT := W#16#0;
   S702_WELD_BUFF_DATA10.RBT9_BT_CODE_NO := W#16#0;
   S702_WELD_BUFF_DATA10.RBT9_WELD_COUNT := W#16#0;
   S702_WELD_BUFF_DATA10.RBT10_BT_CODE_NO := W#16#0;
   S702_WELD_BUFF_DATA10.RBT10_WELD_COUNT := W#16#0;
   S702_WELD_BUFF_DATA10.RBT11_BT_CODE_NO := W#16#0;
   S702_WELD_BUFF_DATA10.RBT11_WELD_COUNT := W#16#0;
   S702_WELD_BUFF_DATA10.RBT12_BT_CODE_NO := W#16#0;
   S702_WELD_BUFF_DATA10.RBT12_WELD_COUNT := W#16#0;
   S702_WELD_BUFF_DATA10.RBT13_BT_CODE_NO := W#16#0;
   S702_WELD_BUFF_DATA10.RBT13_WELD_COUNT := W#16#0;
   S702_WELD_BUFF_DATA10.RBT14_BT_CODE_NO := W#16#0;
   S702_WELD_BUFF_DATA10.RBT14_WELD_COUNT := W#16#0;
   S702_WELD_BUFF_DATA10.RBT15_BT_CODE_NO := W#16#0;
   S702_WELD_BUFF_DATA10.RBT15_WELD_COUNT := W#16#0;
   S702_WELD_BUFF_DATA10.RBT16_BT_CODE_NO := W#16#0;
   S702_WELD_BUFF_DATA10.RBT16_WELD_COUNT := W#16#0;
   S702_WELD_BUFF_DATA10.RBT17_BT_CODE_NO := W#16#0;
   S702_WELD_BUFF_DATA10.RBT17_WELD_COUNT := W#16#0;
   S702_WELD_BUFF_DATA10.RBT18_BT_CODE_NO := W#16#0;
   S702_WELD_BUFF_DATA10.RBT18_WELD_COUNT := W#16#0;
   S702_WELD_BUFF_DATA10.RBT19_BT_CODE_NO := W#16#0;
   S702_WELD_BUFF_DATA10.RBT19_WELD_COUNT := W#16#0;
   S702_WELD_BUFF_DATA10.RBT20_BT_CODE_NO := W#16#0;
   S702_WELD_BUFF_DATA10.RBT20_WELD_COUNT := W#16#0;
   S702_WELD_BUFF_DATA10.RBT21_BT_CODE_NO := W#16#0;
   S702_WELD_BUFF_DATA10.RBT21_WELD_COUNT := W#16#0;
   S702_WELD_BUFF_DATA10.RBT22_BT_CODE_NO := W#16#0;
   S702_WELD_BUFF_DATA10.RBT22_WELD_COUNT := W#16#0;
   S702_WELD_BUFF_DATA10.RBT23_BT_CODE_NO := W#16#0;
   S702_WELD_BUFF_DATA10.RBT23_WELD_COUNT := W#16#0;
   S702_WELD_BUFF_DATA10.RBT24_BT_CODE_NO := W#16#0;
   S702_WELD_BUFF_DATA10.RBT24_WELD_COUNT := W#16#0;
   S702_WELD_BUFF_DATA10.WELD_DETERMINES_RESULT := W#16#0;
   S702_WELD_BUFF_DATA10.WELD_CHECK_SUM := W#16#0;
   S702_WELD_BUFF_DATA10.SPARE1 := W#16#0;
   S703_WELD_BUFF_DATA1.STATION_MAIN := W#16#0;
   S703_WELD_BUFF_DATA1.DISTINCTION_LH_RH := W#16#0;
   S703_WELD_BUFF_DATA1.STAION_NUMBER := W#16#0;
   S703_WELD_BUFF_DATA1.VIN_NUMBER1 := W#16#0;
   S703_WELD_BUFF_DATA1.VIN_NUMBER2 := W#16#0;
   S703_WELD_BUFF_DATA1.VIN_NUMBER3 := W#16#0;
   S703_WELD_BUFF_DATA1.VIN_NUMBER4 := W#16#0;
   S703_WELD_BUFF_DATA1.SEQ_NUMBER1 := W#16#0;
   S703_WELD_BUFF_DATA1.SEQ_NUMBER2 := W#16#0;
   S703_WELD_BUFF_DATA1.RBT1_BT_CODE_NO := W#16#0;
   S703_WELD_BUFF_DATA1.RBT1_WELD_COUNT := W#16#0;
   S703_WELD_BUFF_DATA1.RBT2_BT_CODE_NO := W#16#0;
   S703_WELD_BUFF_DATA1.RBT2_WELD_COUNT := W#16#0;
   S703_WELD_BUFF_DATA1.RBT3_BT_CODE_NO := W#16#0;
   S703_WELD_BUFF_DATA1.RBT3_WELD_COUNT := W#16#0;
   S703_WELD_BUFF_DATA1.RBT4_BT_CODE_NO := W#16#0;
   S703_WELD_BUFF_DATA1.RBT4_WELD_COUNT := W#16#0;
   S703_WELD_BUFF_DATA1.RBT5_BT_CODE_NO := W#16#0;
   S703_WELD_BUFF_DATA1.RBT5_WELD_COUNT := W#16#0;
   S703_WELD_BUFF_DATA1.RBT6_BT_CODE_NO := W#16#0;
   S703_WELD_BUFF_DATA1.RBT6_WELD_COUNT := W#16#0;
   S703_WELD_BUFF_DATA1.RBT7_BT_CODE_NO := W#16#0;
   S703_WELD_BUFF_DATA1.RBT7_WELD_COUNT := W#16#0;
   S703_WELD_BUFF_DATA1.RBT8_BT_CODE_NO := W#16#0;
   S703_WELD_BUFF_DATA1.RBT8_WELD_COUNT := W#16#0;
   S703_WELD_BUFF_DATA1.RBT9_BT_CODE_NO := W#16#0;
   S703_WELD_BUFF_DATA1.RBT9_WELD_COUNT := W#16#0;
   S703_WELD_BUFF_DATA1.RBT10_BT_CODE_NO := W#16#0;
   S703_WELD_BUFF_DATA1.RBT10_WELD_COUNT := W#16#0;
   S703_WELD_BUFF_DATA1.RBT11_BT_CODE_NO := W#16#0;
   S703_WELD_BUFF_DATA1.RBT11_WELD_COUNT := W#16#0;
   S703_WELD_BUFF_DATA1.RBT12_BT_CODE_NO := W#16#0;
   S703_WELD_BUFF_DATA1.RBT12_WELD_COUNT := W#16#0;
   S703_WELD_BUFF_DATA1.RBT13_BT_CODE_NO := W#16#0;
   S703_WELD_BUFF_DATA1.RBT13_WELD_COUNT := W#16#0;
   S703_WELD_BUFF_DATA1.RBT14_BT_CODE_NO := W#16#0;
   S703_WELD_BUFF_DATA1.RBT14_WELD_COUNT := W#16#0;
   S703_WELD_BUFF_DATA1.RBT15_BT_CODE_NO := W#16#0;
   S703_WELD_BUFF_DATA1.RBT15_WELD_COUNT := W#16#0;
   S703_WELD_BUFF_DATA1.RBT16_BT_CODE_NO := W#16#0;
   S703_WELD_BUFF_DATA1.RBT16_WELD_COUNT := W#16#0;
   S703_WELD_BUFF_DATA1.RBT17_BT_CODE_NO := W#16#0;
   S703_WELD_BUFF_DATA1.RBT17_WELD_COUNT := W#16#0;
   S703_WELD_BUFF_DATA1.RBT18_BT_CODE_NO := W#16#0;
   S703_WELD_BUFF_DATA1.RBT18_WELD_COUNT := W#16#0;
   S703_WELD_BUFF_DATA1.RBT19_BT_CODE_NO := W#16#0;
   S703_WELD_BUFF_DATA1.RBT19_WELD_COUNT := W#16#0;
   S703_WELD_BUFF_DATA1.RBT20_BT_CODE_NO := W#16#0;
   S703_WELD_BUFF_DATA1.RBT20_WELD_COUNT := W#16#0;
   S703_WELD_BUFF_DATA1.RBT21_BT_CODE_NO := W#16#0;
   S703_WELD_BUFF_DATA1.RBT21_WELD_COUNT := W#16#0;
   S703_WELD_BUFF_DATA1.RBT22_BT_CODE_NO := W#16#0;
   S703_WELD_BUFF_DATA1.RBT22_WELD_COUNT := W#16#0;
   S703_WELD_BUFF_DATA1.RBT23_BT_CODE_NO := W#16#0;
   S703_WELD_BUFF_DATA1.RBT23_WELD_COUNT := W#16#0;
   S703_WELD_BUFF_DATA1.RBT24_BT_CODE_NO := W#16#0;
   S703_WELD_BUFF_DATA1.RBT24_WELD_COUNT := W#16#0;
   S703_WELD_BUFF_DATA1.WELD_DETERMINES_RESULT := W#16#0;
   S703_WELD_BUFF_DATA1.WELD_CHECK_SUM := W#16#0;
   S703_WELD_BUFF_DATA1.SPARE1 := W#16#0;
   S703_WELD_BUFF_DATA2.STATION_MAIN := W#16#0;
   S703_WELD_BUFF_DATA2.DISTINCTION_LH_RH := W#16#0;
   S703_WELD_BUFF_DATA2.STAION_NUMBER := W#16#0;
   S703_WELD_BUFF_DATA2.VIN_NUMBER1 := W#16#0;
   S703_WELD_BUFF_DATA2.VIN_NUMBER2 := W#16#0;
   S703_WELD_BUFF_DATA2.VIN_NUMBER3 := W#16#0;
   S703_WELD_BUFF_DATA2.VIN_NUMBER4 := W#16#0;
   S703_WELD_BUFF_DATA2.SEQ_NUMBER1 := W#16#0;
   S703_WELD_BUFF_DATA2.SEQ_NUMBER2 := W#16#0;
   S703_WELD_BUFF_DATA2.RBT1_BT_CODE_NO := W#16#0;
   S703_WELD_BUFF_DATA2.RBT1_WELD_COUNT := W#16#0;
   S703_WELD_BUFF_DATA2.RBT2_BT_CODE_NO := W#16#0;
   S703_WELD_BUFF_DATA2.RBT2_WELD_COUNT := W#16#0;
   S703_WELD_BUFF_DATA2.RBT3_BT_CODE_NO := W#16#0;
   S703_WELD_BUFF_DATA2.RBT3_WELD_COUNT := W#16#0;
   S703_WELD_BUFF_DATA2.RBT4_BT_CODE_NO := W#16#0;
   S703_WELD_BUFF_DATA2.RBT4_WELD_COUNT := W#16#0;
   S703_WELD_BUFF_DATA2.RBT5_BT_CODE_NO := W#16#0;
   S703_WELD_BUFF_DATA2.RBT5_WELD_COUNT := W#16#0;
   S703_WELD_BUFF_DATA2.RBT6_BT_CODE_NO := W#16#0;
   S703_WELD_BUFF_DATA2.RBT6_WELD_COUNT := W#16#0;
   S703_WELD_BUFF_DATA2.RBT7_BT_CODE_NO := W#16#0;
   S703_WELD_BUFF_DATA2.RBT7_WELD_COUNT := W#16#0;
   S703_WELD_BUFF_DATA2.RBT8_BT_CODE_NO := W#16#0;
   S703_WELD_BUFF_DATA2.RBT8_WELD_COUNT := W#16#0;
   S703_WELD_BUFF_DATA2.RBT9_BT_CODE_NO := W#16#0;
   S703_WELD_BUFF_DATA2.RBT9_WELD_COUNT := W#16#0;
   S703_WELD_BUFF_DATA2.RBT10_BT_CODE_NO := W#16#0;
   S703_WELD_BUFF_DATA2.RBT10_WELD_COUNT := W#16#0;
   S703_WELD_BUFF_DATA2.RBT11_BT_CODE_NO := W#16#0;
   S703_WELD_BUFF_DATA2.RBT11_WELD_COUNT := W#16#0;
   S703_WELD_BUFF_DATA2.RBT12_BT_CODE_NO := W#16#0;
   S703_WELD_BUFF_DATA2.RBT12_WELD_COUNT := W#16#0;
   S703_WELD_BUFF_DATA2.RBT13_BT_CODE_NO := W#16#0;
   S703_WELD_BUFF_DATA2.RBT13_WELD_COUNT := W#16#0;
   S703_WELD_BUFF_DATA2.RBT14_BT_CODE_NO := W#16#0;
   S703_WELD_BUFF_DATA2.RBT14_WELD_COUNT := W#16#0;
   S703_WELD_BUFF_DATA2.RBT15_BT_CODE_NO := W#16#0;
   S703_WELD_BUFF_DATA2.RBT15_WELD_COUNT := W#16#0;
   S703_WELD_BUFF_DATA2.RBT16_BT_CODE_NO := W#16#0;
   S703_WELD_BUFF_DATA2.RBT16_WELD_COUNT := W#16#0;
   S703_WELD_BUFF_DATA2.RBT17_BT_CODE_NO := W#16#0;
   S703_WELD_BUFF_DATA2.RBT17_WELD_COUNT := W#16#0;
   S703_WELD_BUFF_DATA2.RBT18_BT_CODE_NO := W#16#0;
   S703_WELD_BUFF_DATA2.RBT18_WELD_COUNT := W#16#0;
   S703_WELD_BUFF_DATA2.RBT19_BT_CODE_NO := W#16#0;
   S703_WELD_BUFF_DATA2.RBT19_WELD_COUNT := W#16#0;
   S703_WELD_BUFF_DATA2.RBT20_BT_CODE_NO := W#16#0;
   S703_WELD_BUFF_DATA2.RBT20_WELD_COUNT := W#16#0;
   S703_WELD_BUFF_DATA2.RBT21_BT_CODE_NO := W#16#0;
   S703_WELD_BUFF_DATA2.RBT21_WELD_COUNT := W#16#0;
   S703_WELD_BUFF_DATA2.RBT22_BT_CODE_NO := W#16#0;
   S703_WELD_BUFF_DATA2.RBT22_WELD_COUNT := W#16#0;
   S703_WELD_BUFF_DATA2.RBT23_BT_CODE_NO := W#16#0;
   S703_WELD_BUFF_DATA2.RBT23_WELD_COUNT := W#16#0;
   S703_WELD_BUFF_DATA2.RBT24_BT_CODE_NO := W#16#0;
   S703_WELD_BUFF_DATA2.RBT24_WELD_COUNT := W#16#0;
   S703_WELD_BUFF_DATA2.WELD_DETERMINES_RESULT := W#16#0;
   S703_WELD_BUFF_DATA2.WELD_CHECK_SUM := W#16#0;
   S703_WELD_BUFF_DATA2.SPARE1 := W#16#0;
   S703_WELD_BUFF_DATA3.STATION_MAIN := W#16#0;
   S703_WELD_BUFF_DATA3.DISTINCTION_LH_RH := W#16#0;
   S703_WELD_BUFF_DATA3.STAION_NUMBER := W#16#0;
   S703_WELD_BUFF_DATA3.VIN_NUMBER1 := W#16#0;
   S703_WELD_BUFF_DATA3.VIN_NUMBER2 := W#16#0;
   S703_WELD_BUFF_DATA3.VIN_NUMBER3 := W#16#0;
   S703_WELD_BUFF_DATA3.VIN_NUMBER4 := W#16#0;
   S703_WELD_BUFF_DATA3.SEQ_NUMBER1 := W#16#0;
   S703_WELD_BUFF_DATA3.SEQ_NUMBER2 := W#16#0;
   S703_WELD_BUFF_DATA3.RBT1_BT_CODE_NO := W#16#0;
   S703_WELD_BUFF_DATA3.RBT1_WELD_COUNT := W#16#0;
   S703_WELD_BUFF_DATA3.RBT2_BT_CODE_NO := W#16#0;
   S703_WELD_BUFF_DATA3.RBT2_WELD_COUNT := W#16#0;
   S703_WELD_BUFF_DATA3.RBT3_BT_CODE_NO := W#16#0;
   S703_WELD_BUFF_DATA3.RBT3_WELD_COUNT := W#16#0;
   S703_WELD_BUFF_DATA3.RBT4_BT_CODE_NO := W#16#0;
   S703_WELD_BUFF_DATA3.RBT4_WELD_COUNT := W#16#0;
   S703_WELD_BUFF_DATA3.RBT5_BT_CODE_NO := W#16#0;
   S703_WELD_BUFF_DATA3.RBT5_WELD_COUNT := W#16#0;
   S703_WELD_BUFF_DATA3.RBT6_BT_CODE_NO := W#16#0;
   S703_WELD_BUFF_DATA3.RBT6_WELD_COUNT := W#16#0;
   S703_WELD_BUFF_DATA3.RBT7_BT_CODE_NO := W#16#0;
   S703_WELD_BUFF_DATA3.RBT7_WELD_COUNT := W#16#0;
   S703_WELD_BUFF_DATA3.RBT8_BT_CODE_NO := W#16#0;
   S703_WELD_BUFF_DATA3.RBT8_WELD_COUNT := W#16#0;
   S703_WELD_BUFF_DATA3.RBT9_BT_CODE_NO := W#16#0;
   S703_WELD_BUFF_DATA3.RBT9_WELD_COUNT := W#16#0;
   S703_WELD_BUFF_DATA3.RBT10_BT_CODE_NO := W#16#0;
   S703_WELD_BUFF_DATA3.RBT10_WELD_COUNT := W#16#0;
   S703_WELD_BUFF_DATA3.RBT11_BT_CODE_NO := W#16#0;
   S703_WELD_BUFF_DATA3.RBT11_WELD_COUNT := W#16#0;
   S703_WELD_BUFF_DATA3.RBT12_BT_CODE_NO := W#16#0;
   S703_WELD_BUFF_DATA3.RBT12_WELD_COUNT := W#16#0;
   S703_WELD_BUFF_DATA3.RBT13_BT_CODE_NO := W#16#0;
   S703_WELD_BUFF_DATA3.RBT13_WELD_COUNT := W#16#0;
   S703_WELD_BUFF_DATA3.RBT14_BT_CODE_NO := W#16#0;
   S703_WELD_BUFF_DATA3.RBT14_WELD_COUNT := W#16#0;
   S703_WELD_BUFF_DATA3.RBT15_BT_CODE_NO := W#16#0;
   S703_WELD_BUFF_DATA3.RBT15_WELD_COUNT := W#16#0;
   S703_WELD_BUFF_DATA3.RBT16_BT_CODE_NO := W#16#0;
   S703_WELD_BUFF_DATA3.RBT16_WELD_COUNT := W#16#0;
   S703_WELD_BUFF_DATA3.RBT17_BT_CODE_NO := W#16#0;
   S703_WELD_BUFF_DATA3.RBT17_WELD_COUNT := W#16#0;
   S703_WELD_BUFF_DATA3.RBT18_BT_CODE_NO := W#16#0;
   S703_WELD_BUFF_DATA3.RBT18_WELD_COUNT := W#16#0;
   S703_WELD_BUFF_DATA3.RBT19_BT_CODE_NO := W#16#0;
   S703_WELD_BUFF_DATA3.RBT19_WELD_COUNT := W#16#0;
   S703_WELD_BUFF_DATA3.RBT20_BT_CODE_NO := W#16#0;
   S703_WELD_BUFF_DATA3.RBT20_WELD_COUNT := W#16#0;
   S703_WELD_BUFF_DATA3.RBT21_BT_CODE_NO := W#16#0;
   S703_WELD_BUFF_DATA3.RBT21_WELD_COUNT := W#16#0;
   S703_WELD_BUFF_DATA3.RBT22_BT_CODE_NO := W#16#0;
   S703_WELD_BUFF_DATA3.RBT22_WELD_COUNT := W#16#0;
   S703_WELD_BUFF_DATA3.RBT23_BT_CODE_NO := W#16#0;
   S703_WELD_BUFF_DATA3.RBT23_WELD_COUNT := W#16#0;
   S703_WELD_BUFF_DATA3.RBT24_BT_CODE_NO := W#16#0;
   S703_WELD_BUFF_DATA3.RBT24_WELD_COUNT := W#16#0;
   S703_WELD_BUFF_DATA3.WELD_DETERMINES_RESULT := W#16#0;
   S703_WELD_BUFF_DATA3.WELD_CHECK_SUM := W#16#0;
   S703_WELD_BUFF_DATA3.SPARE1 := W#16#0;
   S703_WELD_BUFF_DATA4.STATION_MAIN := W#16#0;
   S703_WELD_BUFF_DATA4.DISTINCTION_LH_RH := W#16#0;
   S703_WELD_BUFF_DATA4.STAION_NUMBER := W#16#0;
   S703_WELD_BUFF_DATA4.VIN_NUMBER1 := W#16#0;
   S703_WELD_BUFF_DATA4.VIN_NUMBER2 := W#16#0;
   S703_WELD_BUFF_DATA4.VIN_NUMBER3 := W#16#0;
   S703_WELD_BUFF_DATA4.VIN_NUMBER4 := W#16#0;
   S703_WELD_BUFF_DATA4.SEQ_NUMBER1 := W#16#0;
   S703_WELD_BUFF_DATA4.SEQ_NUMBER2 := W#16#0;
   S703_WELD_BUFF_DATA4.RBT1_BT_CODE_NO := W#16#0;
   S703_WELD_BUFF_DATA4.RBT1_WELD_COUNT := W#16#0;
   S703_WELD_BUFF_DATA4.RBT2_BT_CODE_NO := W#16#0;
   S703_WELD_BUFF_DATA4.RBT2_WELD_COUNT := W#16#0;
   S703_WELD_BUFF_DATA4.RBT3_BT_CODE_NO := W#16#0;
   S703_WELD_BUFF_DATA4.RBT3_WELD_COUNT := W#16#0;
   S703_WELD_BUFF_DATA4.RBT4_BT_CODE_NO := W#16#0;
   S703_WELD_BUFF_DATA4.RBT4_WELD_COUNT := W#16#0;
   S703_WELD_BUFF_DATA4.RBT5_BT_CODE_NO := W#16#0;
   S703_WELD_BUFF_DATA4.RBT5_WELD_COUNT := W#16#0;
   S703_WELD_BUFF_DATA4.RBT6_BT_CODE_NO := W#16#0;
   S703_WELD_BUFF_DATA4.RBT6_WELD_COUNT := W#16#0;
   S703_WELD_BUFF_DATA4.RBT7_BT_CODE_NO := W#16#0;
   S703_WELD_BUFF_DATA4.RBT7_WELD_COUNT := W#16#0;
   S703_WELD_BUFF_DATA4.RBT8_BT_CODE_NO := W#16#0;
   S703_WELD_BUFF_DATA4.RBT8_WELD_COUNT := W#16#0;
   S703_WELD_BUFF_DATA4.RBT9_BT_CODE_NO := W#16#0;
   S703_WELD_BUFF_DATA4.RBT9_WELD_COUNT := W#16#0;
   S703_WELD_BUFF_DATA4.RBT10_BT_CODE_NO := W#16#0;
   S703_WELD_BUFF_DATA4.RBT10_WELD_COUNT := W#16#0;
   S703_WELD_BUFF_DATA4.RBT11_BT_CODE_NO := W#16#0;
   S703_WELD_BUFF_DATA4.RBT11_WELD_COUNT := W#16#0;
   S703_WELD_BUFF_DATA4.RBT12_BT_CODE_NO := W#16#0;
   S703_WELD_BUFF_DATA4.RBT12_WELD_COUNT := W#16#0;
   S703_WELD_BUFF_DATA4.RBT13_BT_CODE_NO := W#16#0;
   S703_WELD_BUFF_DATA4.RBT13_WELD_COUNT := W#16#0;
   S703_WELD_BUFF_DATA4.RBT14_BT_CODE_NO := W#16#0;
   S703_WELD_BUFF_DATA4.RBT14_WELD_COUNT := W#16#0;
   S703_WELD_BUFF_DATA4.RBT15_BT_CODE_NO := W#16#0;
   S703_WELD_BUFF_DATA4.RBT15_WELD_COUNT := W#16#0;
   S703_WELD_BUFF_DATA4.RBT16_BT_CODE_NO := W#16#0;
   S703_WELD_BUFF_DATA4.RBT16_WELD_COUNT := W#16#0;
   S703_WELD_BUFF_DATA4.RBT17_BT_CODE_NO := W#16#0;
   S703_WELD_BUFF_DATA4.RBT17_WELD_COUNT := W#16#0;
   S703_WELD_BUFF_DATA4.RBT18_BT_CODE_NO := W#16#0;
   S703_WELD_BUFF_DATA4.RBT18_WELD_COUNT := W#16#0;
   S703_WELD_BUFF_DATA4.RBT19_BT_CODE_NO := W#16#0;
   S703_WELD_BUFF_DATA4.RBT19_WELD_COUNT := W#16#0;
   S703_WELD_BUFF_DATA4.RBT20_BT_CODE_NO := W#16#0;
   S703_WELD_BUFF_DATA4.RBT20_WELD_COUNT := W#16#0;
   S703_WELD_BUFF_DATA4.RBT21_BT_CODE_NO := W#16#0;
   S703_WELD_BUFF_DATA4.RBT21_WELD_COUNT := W#16#0;
   S703_WELD_BUFF_DATA4.RBT22_BT_CODE_NO := W#16#0;
   S703_WELD_BUFF_DATA4.RBT22_WELD_COUNT := W#16#0;
   S703_WELD_BUFF_DATA4.RBT23_BT_CODE_NO := W#16#0;
   S703_WELD_BUFF_DATA4.RBT23_WELD_COUNT := W#16#0;
   S703_WELD_BUFF_DATA4.RBT24_BT_CODE_NO := W#16#0;
   S703_WELD_BUFF_DATA4.RBT24_WELD_COUNT := W#16#0;
   S703_WELD_BUFF_DATA4.WELD_DETERMINES_RESULT := W#16#0;
   S703_WELD_BUFF_DATA4.WELD_CHECK_SUM := W#16#0;
   S703_WELD_BUFF_DATA4.SPARE1 := W#16#0;
   S703_WELD_BUFF_DATA5.STATION_MAIN := W#16#0;
   S703_WELD_BUFF_DATA5.DISTINCTION_LH_RH := W#16#0;
   S703_WELD_BUFF_DATA5.STAION_NUMBER := W#16#0;
   S703_WELD_BUFF_DATA5.VIN_NUMBER1 := W#16#0;
   S703_WELD_BUFF_DATA5.VIN_NUMBER2 := W#16#0;
   S703_WELD_BUFF_DATA5.VIN_NUMBER3 := W#16#0;
   S703_WELD_BUFF_DATA5.VIN_NUMBER4 := W#16#0;
   S703_WELD_BUFF_DATA5.SEQ_NUMBER1 := W#16#0;
   S703_WELD_BUFF_DATA5.SEQ_NUMBER2 := W#16#0;
   S703_WELD_BUFF_DATA5.RBT1_BT_CODE_NO := W#16#0;
   S703_WELD_BUFF_DATA5.RBT1_WELD_COUNT := W#16#0;
   S703_WELD_BUFF_DATA5.RBT2_BT_CODE_NO := W#16#0;
   S703_WELD_BUFF_DATA5.RBT2_WELD_COUNT := W#16#0;
   S703_WELD_BUFF_DATA5.RBT3_BT_CODE_NO := W#16#0;
   S703_WELD_BUFF_DATA5.RBT3_WELD_COUNT := W#16#0;
   S703_WELD_BUFF_DATA5.RBT4_BT_CODE_NO := W#16#0;
   S703_WELD_BUFF_DATA5.RBT4_WELD_COUNT := W#16#0;
   S703_WELD_BUFF_DATA5.RBT5_BT_CODE_NO := W#16#0;
   S703_WELD_BUFF_DATA5.RBT5_WELD_COUNT := W#16#0;
   S703_WELD_BUFF_DATA5.RBT6_BT_CODE_NO := W#16#0;
   S703_WELD_BUFF_DATA5.RBT6_WELD_COUNT := W#16#0;
   S703_WELD_BUFF_DATA5.RBT7_BT_CODE_NO := W#16#0;
   S703_WELD_BUFF_DATA5.RBT7_WELD_COUNT := W#16#0;
   S703_WELD_BUFF_DATA5.RBT8_BT_CODE_NO := W#16#0;
   S703_WELD_BUFF_DATA5.RBT8_WELD_COUNT := W#16#0;
   S703_WELD_BUFF_DATA5.RBT9_BT_CODE_NO := W#16#0;
   S703_WELD_BUFF_DATA5.RBT9_WELD_COUNT := W#16#0;
   S703_WELD_BUFF_DATA5.RBT10_BT_CODE_NO := W#16#0;
   S703_WELD_BUFF_DATA5.RBT10_WELD_COUNT := W#16#0;
   S703_WELD_BUFF_DATA5.RBT11_BT_CODE_NO := W#16#0;
   S703_WELD_BUFF_DATA5.RBT11_WELD_COUNT := W#16#0;
   S703_WELD_BUFF_DATA5.RBT12_BT_CODE_NO := W#16#0;
   S703_WELD_BUFF_DATA5.RBT12_WELD_COUNT := W#16#0;
   S703_WELD_BUFF_DATA5.RBT13_BT_CODE_NO := W#16#0;
   S703_WELD_BUFF_DATA5.RBT13_WELD_COUNT := W#16#0;
   S703_WELD_BUFF_DATA5.RBT14_BT_CODE_NO := W#16#0;
   S703_WELD_BUFF_DATA5.RBT14_WELD_COUNT := W#16#0;
   S703_WELD_BUFF_DATA5.RBT15_BT_CODE_NO := W#16#0;
   S703_WELD_BUFF_DATA5.RBT15_WELD_COUNT := W#16#0;
   S703_WELD_BUFF_DATA5.RBT16_BT_CODE_NO := W#16#0;
   S703_WELD_BUFF_DATA5.RBT16_WELD_COUNT := W#16#0;
   S703_WELD_BUFF_DATA5.RBT17_BT_CODE_NO := W#16#0;
   S703_WELD_BUFF_DATA5.RBT17_WELD_COUNT := W#16#0;
   S703_WELD_BUFF_DATA5.RBT18_BT_CODE_NO := W#16#0;
   S703_WELD_BUFF_DATA5.RBT18_WELD_COUNT := W#16#0;
   S703_WELD_BUFF_DATA5.RBT19_BT_CODE_NO := W#16#0;
   S703_WELD_BUFF_DATA5.RBT19_WELD_COUNT := W#16#0;
   S703_WELD_BUFF_DATA5.RBT20_BT_CODE_NO := W#16#0;
   S703_WELD_BUFF_DATA5.RBT20_WELD_COUNT := W#16#0;
   S703_WELD_BUFF_DATA5.RBT21_BT_CODE_NO := W#16#0;
   S703_WELD_BUFF_DATA5.RBT21_WELD_COUNT := W#16#0;
   S703_WELD_BUFF_DATA5.RBT22_BT_CODE_NO := W#16#0;
   S703_WELD_BUFF_DATA5.RBT22_WELD_COUNT := W#16#0;
   S703_WELD_BUFF_DATA5.RBT23_BT_CODE_NO := W#16#0;
   S703_WELD_BUFF_DATA5.RBT23_WELD_COUNT := W#16#0;
   S703_WELD_BUFF_DATA5.RBT24_BT_CODE_NO := W#16#0;
   S703_WELD_BUFF_DATA5.RBT24_WELD_COUNT := W#16#0;
   S703_WELD_BUFF_DATA5.WELD_DETERMINES_RESULT := W#16#0;
   S703_WELD_BUFF_DATA5.WELD_CHECK_SUM := W#16#0;
   S703_WELD_BUFF_DATA5.SPARE1 := W#16#0;
   S703_WELD_BUFF_DATA6.STATION_MAIN := W#16#0;
   S703_WELD_BUFF_DATA6.DISTINCTION_LH_RH := W#16#0;
   S703_WELD_BUFF_DATA6.STAION_NUMBER := W#16#0;
   S703_WELD_BUFF_DATA6.VIN_NUMBER1 := W#16#0;
   S703_WELD_BUFF_DATA6.VIN_NUMBER2 := W#16#0;
   S703_WELD_BUFF_DATA6.VIN_NUMBER3 := W#16#0;
   S703_WELD_BUFF_DATA6.VIN_NUMBER4 := W#16#0;
   S703_WELD_BUFF_DATA6.SEQ_NUMBER1 := W#16#0;
   S703_WELD_BUFF_DATA6.SEQ_NUMBER2 := W#16#0;
   S703_WELD_BUFF_DATA6.RBT1_BT_CODE_NO := W#16#0;
   S703_WELD_BUFF_DATA6.RBT1_WELD_COUNT := W#16#0;
   S703_WELD_BUFF_DATA6.RBT2_BT_CODE_NO := W#16#0;
   S703_WELD_BUFF_DATA6.RBT2_WELD_COUNT := W#16#0;
   S703_WELD_BUFF_DATA6.RBT3_BT_CODE_NO := W#16#0;
   S703_WELD_BUFF_DATA6.RBT3_WELD_COUNT := W#16#0;
   S703_WELD_BUFF_DATA6.RBT4_BT_CODE_NO := W#16#0;
   S703_WELD_BUFF_DATA6.RBT4_WELD_COUNT := W#16#0;
   S703_WELD_BUFF_DATA6.RBT5_BT_CODE_NO := W#16#0;
   S703_WELD_BUFF_DATA6.RBT5_WELD_COUNT := W#16#0;
   S703_WELD_BUFF_DATA6.RBT6_BT_CODE_NO := W#16#0;
   S703_WELD_BUFF_DATA6.RBT6_WELD_COUNT := W#16#0;
   S703_WELD_BUFF_DATA6.RBT7_BT_CODE_NO := W#16#0;
   S703_WELD_BUFF_DATA6.RBT7_WELD_COUNT := W#16#0;
   S703_WELD_BUFF_DATA6.RBT8_BT_CODE_NO := W#16#0;
   S703_WELD_BUFF_DATA6.RBT8_WELD_COUNT := W#16#0;
   S703_WELD_BUFF_DATA6.RBT9_BT_CODE_NO := W#16#0;
   S703_WELD_BUFF_DATA6.RBT9_WELD_COUNT := W#16#0;
   S703_WELD_BUFF_DATA6.RBT10_BT_CODE_NO := W#16#0;
   S703_WELD_BUFF_DATA6.RBT10_WELD_COUNT := W#16#0;
   S703_WELD_BUFF_DATA6.RBT11_BT_CODE_NO := W#16#0;
   S703_WELD_BUFF_DATA6.RBT11_WELD_COUNT := W#16#0;
   S703_WELD_BUFF_DATA6.RBT12_BT_CODE_NO := W#16#0;
   S703_WELD_BUFF_DATA6.RBT12_WELD_COUNT := W#16#0;
   S703_WELD_BUFF_DATA6.RBT13_BT_CODE_NO := W#16#0;
   S703_WELD_BUFF_DATA6.RBT13_WELD_COUNT := W#16#0;
   S703_WELD_BUFF_DATA6.RBT14_BT_CODE_NO := W#16#0;
   S703_WELD_BUFF_DATA6.RBT14_WELD_COUNT := W#16#0;
   S703_WELD_BUFF_DATA6.RBT15_BT_CODE_NO := W#16#0;
   S703_WELD_BUFF_DATA6.RBT15_WELD_COUNT := W#16#0;
   S703_WELD_BUFF_DATA6.RBT16_BT_CODE_NO := W#16#0;
   S703_WELD_BUFF_DATA6.RBT16_WELD_COUNT := W#16#0;
   S703_WELD_BUFF_DATA6.RBT17_BT_CODE_NO := W#16#0;
   S703_WELD_BUFF_DATA6.RBT17_WELD_COUNT := W#16#0;
   S703_WELD_BUFF_DATA6.RBT18_BT_CODE_NO := W#16#0;
   S703_WELD_BUFF_DATA6.RBT18_WELD_COUNT := W#16#0;
   S703_WELD_BUFF_DATA6.RBT19_BT_CODE_NO := W#16#0;
   S703_WELD_BUFF_DATA6.RBT19_WELD_COUNT := W#16#0;
   S703_WELD_BUFF_DATA6.RBT20_BT_CODE_NO := W#16#0;
   S703_WELD_BUFF_DATA6.RBT20_WELD_COUNT := W#16#0;
   S703_WELD_BUFF_DATA6.RBT21_BT_CODE_NO := W#16#0;
   S703_WELD_BUFF_DATA6.RBT21_WELD_COUNT := W#16#0;
   S703_WELD_BUFF_DATA6.RBT22_BT_CODE_NO := W#16#0;
   S703_WELD_BUFF_DATA6.RBT22_WELD_COUNT := W#16#0;
   S703_WELD_BUFF_DATA6.RBT23_BT_CODE_NO := W#16#0;
   S703_WELD_BUFF_DATA6.RBT23_WELD_COUNT := W#16#0;
   S703_WELD_BUFF_DATA6.RBT24_BT_CODE_NO := W#16#0;
   S703_WELD_BUFF_DATA6.RBT24_WELD_COUNT := W#16#0;
   S703_WELD_BUFF_DATA6.WELD_DETERMINES_RESULT := W#16#0;
   S703_WELD_BUFF_DATA6.WELD_CHECK_SUM := W#16#0;
   S703_WELD_BUFF_DATA6.SPARE1 := W#16#0;
   S703_WELD_BUFF_DATA7.STATION_MAIN := W#16#0;
   S703_WELD_BUFF_DATA7.DISTINCTION_LH_RH := W#16#0;
   S703_WELD_BUFF_DATA7.STAION_NUMBER := W#16#0;
   S703_WELD_BUFF_DATA7.VIN_NUMBER1 := W#16#0;
   S703_WELD_BUFF_DATA7.VIN_NUMBER2 := W#16#0;
   S703_WELD_BUFF_DATA7.VIN_NUMBER3 := W#16#0;
   S703_WELD_BUFF_DATA7.VIN_NUMBER4 := W#16#0;
   S703_WELD_BUFF_DATA7.SEQ_NUMBER1 := W#16#0;
   S703_WELD_BUFF_DATA7.SEQ_NUMBER2 := W#16#0;
   S703_WELD_BUFF_DATA7.RBT1_BT_CODE_NO := W#16#0;
   S703_WELD_BUFF_DATA7.RBT1_WELD_COUNT := W#16#0;
   S703_WELD_BUFF_DATA7.RBT2_BT_CODE_NO := W#16#0;
   S703_WELD_BUFF_DATA7.RBT2_WELD_COUNT := W#16#0;
   S703_WELD_BUFF_DATA7.RBT3_BT_CODE_NO := W#16#0;
   S703_WELD_BUFF_DATA7.RBT3_WELD_COUNT := W#16#0;
   S703_WELD_BUFF_DATA7.RBT4_BT_CODE_NO := W#16#0;
   S703_WELD_BUFF_DATA7.RBT4_WELD_COUNT := W#16#0;
   S703_WELD_BUFF_DATA7.RBT5_BT_CODE_NO := W#16#0;
   S703_WELD_BUFF_DATA7.RBT5_WELD_COUNT := W#16#0;
   S703_WELD_BUFF_DATA7.RBT6_BT_CODE_NO := W#16#0;
   S703_WELD_BUFF_DATA7.RBT6_WELD_COUNT := W#16#0;
   S703_WELD_BUFF_DATA7.RBT7_BT_CODE_NO := W#16#0;
   S703_WELD_BUFF_DATA7.RBT7_WELD_COUNT := W#16#0;
   S703_WELD_BUFF_DATA7.RBT8_BT_CODE_NO := W#16#0;
   S703_WELD_BUFF_DATA7.RBT8_WELD_COUNT := W#16#0;
   S703_WELD_BUFF_DATA7.RBT9_BT_CODE_NO := W#16#0;
   S703_WELD_BUFF_DATA7.RBT9_WELD_COUNT := W#16#0;
   S703_WELD_BUFF_DATA7.RBT10_BT_CODE_NO := W#16#0;
   S703_WELD_BUFF_DATA7.RBT10_WELD_COUNT := W#16#0;
   S703_WELD_BUFF_DATA7.RBT11_BT_CODE_NO := W#16#0;
   S703_WELD_BUFF_DATA7.RBT11_WELD_COUNT := W#16#0;
   S703_WELD_BUFF_DATA7.RBT12_BT_CODE_NO := W#16#0;
   S703_WELD_BUFF_DATA7.RBT12_WELD_COUNT := W#16#0;
   S703_WELD_BUFF_DATA7.RBT13_BT_CODE_NO := W#16#0;
   S703_WELD_BUFF_DATA7.RBT13_WELD_COUNT := W#16#0;
   S703_WELD_BUFF_DATA7.RBT14_BT_CODE_NO := W#16#0;
   S703_WELD_BUFF_DATA7.RBT14_WELD_COUNT := W#16#0;
   S703_WELD_BUFF_DATA7.RBT15_BT_CODE_NO := W#16#0;
   S703_WELD_BUFF_DATA7.RBT15_WELD_COUNT := W#16#0;
   S703_WELD_BUFF_DATA7.RBT16_BT_CODE_NO := W#16#0;
   S703_WELD_BUFF_DATA7.RBT16_WELD_COUNT := W#16#0;
   S703_WELD_BUFF_DATA7.RBT17_BT_CODE_NO := W#16#0;
   S703_WELD_BUFF_DATA7.RBT17_WELD_COUNT := W#16#0;
   S703_WELD_BUFF_DATA7.RBT18_BT_CODE_NO := W#16#0;
   S703_WELD_BUFF_DATA7.RBT18_WELD_COUNT := W#16#0;
   S703_WELD_BUFF_DATA7.RBT19_BT_CODE_NO := W#16#0;
   S703_WELD_BUFF_DATA7.RBT19_WELD_COUNT := W#16#0;
   S703_WELD_BUFF_DATA7.RBT20_BT_CODE_NO := W#16#0;
   S703_WELD_BUFF_DATA7.RBT20_WELD_COUNT := W#16#0;
   S703_WELD_BUFF_DATA7.RBT21_BT_CODE_NO := W#16#0;
   S703_WELD_BUFF_DATA7.RBT21_WELD_COUNT := W#16#0;
   S703_WELD_BUFF_DATA7.RBT22_BT_CODE_NO := W#16#0;
   S703_WELD_BUFF_DATA7.RBT22_WELD_COUNT := W#16#0;
   S703_WELD_BUFF_DATA7.RBT23_BT_CODE_NO := W#16#0;
   S703_WELD_BUFF_DATA7.RBT23_WELD_COUNT := W#16#0;
   S703_WELD_BUFF_DATA7.RBT24_BT_CODE_NO := W#16#0;
   S703_WELD_BUFF_DATA7.RBT24_WELD_COUNT := W#16#0;
   S703_WELD_BUFF_DATA7.WELD_DETERMINES_RESULT := W#16#0;
   S703_WELD_BUFF_DATA7.WELD_CHECK_SUM := W#16#0;
   S703_WELD_BUFF_DATA7.SPARE1 := W#16#0;
   S703_WELD_BUFF_DATA8.STATION_MAIN := W#16#0;
   S703_WELD_BUFF_DATA8.DISTINCTION_LH_RH := W#16#0;
   S703_WELD_BUFF_DATA8.STAION_NUMBER := W#16#0;
   S703_WELD_BUFF_DATA8.VIN_NUMBER1 := W#16#0;
   S703_WELD_BUFF_DATA8.VIN_NUMBER2 := W#16#0;
   S703_WELD_BUFF_DATA8.VIN_NUMBER3 := W#16#0;
   S703_WELD_BUFF_DATA8.VIN_NUMBER4 := W#16#0;
   S703_WELD_BUFF_DATA8.SEQ_NUMBER1 := W#16#0;
   S703_WELD_BUFF_DATA8.SEQ_NUMBER2 := W#16#0;
   S703_WELD_BUFF_DATA8.RBT1_BT_CODE_NO := W#16#0;
   S703_WELD_BUFF_DATA8.RBT1_WELD_COUNT := W#16#0;
   S703_WELD_BUFF_DATA8.RBT2_BT_CODE_NO := W#16#0;
   S703_WELD_BUFF_DATA8.RBT2_WELD_COUNT := W#16#0;
   S703_WELD_BUFF_DATA8.RBT3_BT_CODE_NO := W#16#0;
   S703_WELD_BUFF_DATA8.RBT3_WELD_COUNT := W#16#0;
   S703_WELD_BUFF_DATA8.RBT4_BT_CODE_NO := W#16#0;
   S703_WELD_BUFF_DATA8.RBT4_WELD_COUNT := W#16#0;
   S703_WELD_BUFF_DATA8.RBT5_BT_CODE_NO := W#16#0;
   S703_WELD_BUFF_DATA8.RBT5_WELD_COUNT := W#16#0;
   S703_WELD_BUFF_DATA8.RBT6_BT_CODE_NO := W#16#0;
   S703_WELD_BUFF_DATA8.RBT6_WELD_COUNT := W#16#0;
   S703_WELD_BUFF_DATA8.RBT7_BT_CODE_NO := W#16#0;
   S703_WELD_BUFF_DATA8.RBT7_WELD_COUNT := W#16#0;
   S703_WELD_BUFF_DATA8.RBT8_BT_CODE_NO := W#16#0;
   S703_WELD_BUFF_DATA8.RBT8_WELD_COUNT := W#16#0;
   S703_WELD_BUFF_DATA8.RBT9_BT_CODE_NO := W#16#0;
   S703_WELD_BUFF_DATA8.RBT9_WELD_COUNT := W#16#0;
   S703_WELD_BUFF_DATA8.RBT10_BT_CODE_NO := W#16#0;
   S703_WELD_BUFF_DATA8.RBT10_WELD_COUNT := W#16#0;
   S703_WELD_BUFF_DATA8.RBT11_BT_CODE_NO := W#16#0;
   S703_WELD_BUFF_DATA8.RBT11_WELD_COUNT := W#16#0;
   S703_WELD_BUFF_DATA8.RBT12_BT_CODE_NO := W#16#0;
   S703_WELD_BUFF_DATA8.RBT12_WELD_COUNT := W#16#0;
   S703_WELD_BUFF_DATA8.RBT13_BT_CODE_NO := W#16#0;
   S703_WELD_BUFF_DATA8.RBT13_WELD_COUNT := W#16#0;
   S703_WELD_BUFF_DATA8.RBT14_BT_CODE_NO := W#16#0;
   S703_WELD_BUFF_DATA8.RBT14_WELD_COUNT := W#16#0;
   S703_WELD_BUFF_DATA8.RBT15_BT_CODE_NO := W#16#0;
   S703_WELD_BUFF_DATA8.RBT15_WELD_COUNT := W#16#0;
   S703_WELD_BUFF_DATA8.RBT16_BT_CODE_NO := W#16#0;
   S703_WELD_BUFF_DATA8.RBT16_WELD_COUNT := W#16#0;
   S703_WELD_BUFF_DATA8.RBT17_BT_CODE_NO := W#16#0;
   S703_WELD_BUFF_DATA8.RBT17_WELD_COUNT := W#16#0;
   S703_WELD_BUFF_DATA8.RBT18_BT_CODE_NO := W#16#0;
   S703_WELD_BUFF_DATA8.RBT18_WELD_COUNT := W#16#0;
   S703_WELD_BUFF_DATA8.RBT19_BT_CODE_NO := W#16#0;
   S703_WELD_BUFF_DATA8.RBT19_WELD_COUNT := W#16#0;
   S703_WELD_BUFF_DATA8.RBT20_BT_CODE_NO := W#16#0;
   S703_WELD_BUFF_DATA8.RBT20_WELD_COUNT := W#16#0;
   S703_WELD_BUFF_DATA8.RBT21_BT_CODE_NO := W#16#0;
   S703_WELD_BUFF_DATA8.RBT21_WELD_COUNT := W#16#0;
   S703_WELD_BUFF_DATA8.RBT22_BT_CODE_NO := W#16#0;
   S703_WELD_BUFF_DATA8.RBT22_WELD_COUNT := W#16#0;
   S703_WELD_BUFF_DATA8.RBT23_BT_CODE_NO := W#16#0;
   S703_WELD_BUFF_DATA8.RBT23_WELD_COUNT := W#16#0;
   S703_WELD_BUFF_DATA8.RBT24_BT_CODE_NO := W#16#0;
   S703_WELD_BUFF_DATA8.RBT24_WELD_COUNT := W#16#0;
   S703_WELD_BUFF_DATA8.WELD_DETERMINES_RESULT := W#16#0;
   S703_WELD_BUFF_DATA8.WELD_CHECK_SUM := W#16#0;
   S703_WELD_BUFF_DATA8.SPARE1 := W#16#0;
   S703_WELD_BUFF_DATA9.STATION_MAIN := W#16#0;
   S703_WELD_BUFF_DATA9.DISTINCTION_LH_RH := W#16#0;
   S703_WELD_BUFF_DATA9.STAION_NUMBER := W#16#0;
   S703_WELD_BUFF_DATA9.VIN_NUMBER1 := W#16#0;
   S703_WELD_BUFF_DATA9.VIN_NUMBER2 := W#16#0;
   S703_WELD_BUFF_DATA9.VIN_NUMBER3 := W#16#0;
   S703_WELD_BUFF_DATA9.VIN_NUMBER4 := W#16#0;
   S703_WELD_BUFF_DATA9.SEQ_NUMBER1 := W#16#0;
   S703_WELD_BUFF_DATA9.SEQ_NUMBER2 := W#16#0;
   S703_WELD_BUFF_DATA9.RBT1_BT_CODE_NO := W#16#0;
   S703_WELD_BUFF_DATA9.RBT1_WELD_COUNT := W#16#0;
   S703_WELD_BUFF_DATA9.RBT2_BT_CODE_NO := W#16#0;
   S703_WELD_BUFF_DATA9.RBT2_WELD_COUNT := W#16#0;
   S703_WELD_BUFF_DATA9.RBT3_BT_CODE_NO := W#16#0;
   S703_WELD_BUFF_DATA9.RBT3_WELD_COUNT := W#16#0;
   S703_WELD_BUFF_DATA9.RBT4_BT_CODE_NO := W#16#0;
   S703_WELD_BUFF_DATA9.RBT4_WELD_COUNT := W#16#0;
   S703_WELD_BUFF_DATA9.RBT5_BT_CODE_NO := W#16#0;
   S703_WELD_BUFF_DATA9.RBT5_WELD_COUNT := W#16#0;
   S703_WELD_BUFF_DATA9.RBT6_BT_CODE_NO := W#16#0;
   S703_WELD_BUFF_DATA9.RBT6_WELD_COUNT := W#16#0;
   S703_WELD_BUFF_DATA9.RBT7_BT_CODE_NO := W#16#0;
   S703_WELD_BUFF_DATA9.RBT7_WELD_COUNT := W#16#0;
   S703_WELD_BUFF_DATA9.RBT8_BT_CODE_NO := W#16#0;
   S703_WELD_BUFF_DATA9.RBT8_WELD_COUNT := W#16#0;
   S703_WELD_BUFF_DATA9.RBT9_BT_CODE_NO := W#16#0;
   S703_WELD_BUFF_DATA9.RBT9_WELD_COUNT := W#16#0;
   S703_WELD_BUFF_DATA9.RBT10_BT_CODE_NO := W#16#0;
   S703_WELD_BUFF_DATA9.RBT10_WELD_COUNT := W#16#0;
   S703_WELD_BUFF_DATA9.RBT11_BT_CODE_NO := W#16#0;
   S703_WELD_BUFF_DATA9.RBT11_WELD_COUNT := W#16#0;
   S703_WELD_BUFF_DATA9.RBT12_BT_CODE_NO := W#16#0;
   S703_WELD_BUFF_DATA9.RBT12_WELD_COUNT := W#16#0;
   S703_WELD_BUFF_DATA9.RBT13_BT_CODE_NO := W#16#0;
   S703_WELD_BUFF_DATA9.RBT13_WELD_COUNT := W#16#0;
   S703_WELD_BUFF_DATA9.RBT14_BT_CODE_NO := W#16#0;
   S703_WELD_BUFF_DATA9.RBT14_WELD_COUNT := W#16#0;
   S703_WELD_BUFF_DATA9.RBT15_BT_CODE_NO := W#16#0;
   S703_WELD_BUFF_DATA9.RBT15_WELD_COUNT := W#16#0;
   S703_WELD_BUFF_DATA9.RBT16_BT_CODE_NO := W#16#0;
   S703_WELD_BUFF_DATA9.RBT16_WELD_COUNT := W#16#0;
   S703_WELD_BUFF_DATA9.RBT17_BT_CODE_NO := W#16#0;
   S703_WELD_BUFF_DATA9.RBT17_WELD_COUNT := W#16#0;
   S703_WELD_BUFF_DATA9.RBT18_BT_CODE_NO := W#16#0;
   S703_WELD_BUFF_DATA9.RBT18_WELD_COUNT := W#16#0;
   S703_WELD_BUFF_DATA9.RBT19_BT_CODE_NO := W#16#0;
   S703_WELD_BUFF_DATA9.RBT19_WELD_COUNT := W#16#0;
   S703_WELD_BUFF_DATA9.RBT20_BT_CODE_NO := W#16#0;
   S703_WELD_BUFF_DATA9.RBT20_WELD_COUNT := W#16#0;
   S703_WELD_BUFF_DATA9.RBT21_BT_CODE_NO := W#16#0;
   S703_WELD_BUFF_DATA9.RBT21_WELD_COUNT := W#16#0;
   S703_WELD_BUFF_DATA9.RBT22_BT_CODE_NO := W#16#0;
   S703_WELD_BUFF_DATA9.RBT22_WELD_COUNT := W#16#0;
   S703_WELD_BUFF_DATA9.RBT23_BT_CODE_NO := W#16#0;
   S703_WELD_BUFF_DATA9.RBT23_WELD_COUNT := W#16#0;
   S703_WELD_BUFF_DATA9.RBT24_BT_CODE_NO := W#16#0;
   S703_WELD_BUFF_DATA9.RBT24_WELD_COUNT := W#16#0;
   S703_WELD_BUFF_DATA9.WELD_DETERMINES_RESULT := W#16#0;
   S703_WELD_BUFF_DATA9.WELD_CHECK_SUM := W#16#0;
   S703_WELD_BUFF_DATA9.SPARE1 := W#16#0;
   S703_WELD_BUFF_DATA10.STATION_MAIN := W#16#0;
   S703_WELD_BUFF_DATA10.DISTINCTION_LH_RH := W#16#0;
   S703_WELD_BUFF_DATA10.STAION_NUMBER := W#16#0;
   S703_WELD_BUFF_DATA10.VIN_NUMBER1 := W#16#0;
   S703_WELD_BUFF_DATA10.VIN_NUMBER2 := W#16#0;
   S703_WELD_BUFF_DATA10.VIN_NUMBER3 := W#16#0;
   S703_WELD_BUFF_DATA10.VIN_NUMBER4 := W#16#0;
   S703_WELD_BUFF_DATA10.SEQ_NUMBER1 := W#16#0;
   S703_WELD_BUFF_DATA10.SEQ_NUMBER2 := W#16#0;
   S703_WELD_BUFF_DATA10.RBT1_BT_CODE_NO := W#16#0;
   S703_WELD_BUFF_DATA10.RBT1_WELD_COUNT := W#16#0;
   S703_WELD_BUFF_DATA10.RBT2_BT_CODE_NO := W#16#0;
   S703_WELD_BUFF_DATA10.RBT2_WELD_COUNT := W#16#0;
   S703_WELD_BUFF_DATA10.RBT3_BT_CODE_NO := W#16#0;
   S703_WELD_BUFF_DATA10.RBT3_WELD_COUNT := W#16#0;
   S703_WELD_BUFF_DATA10.RBT4_BT_CODE_NO := W#16#0;
   S703_WELD_BUFF_DATA10.RBT4_WELD_COUNT := W#16#0;
   S703_WELD_BUFF_DATA10.RBT5_BT_CODE_NO := W#16#0;
   S703_WELD_BUFF_DATA10.RBT5_WELD_COUNT := W#16#0;
   S703_WELD_BUFF_DATA10.RBT6_BT_CODE_NO := W#16#0;
   S703_WELD_BUFF_DATA10.RBT6_WELD_COUNT := W#16#0;
   S703_WELD_BUFF_DATA10.RBT7_BT_CODE_NO := W#16#0;
   S703_WELD_BUFF_DATA10.RBT7_WELD_COUNT := W#16#0;
   S703_WELD_BUFF_DATA10.RBT8_BT_CODE_NO := W#16#0;
   S703_WELD_BUFF_DATA10.RBT8_WELD_COUNT := W#16#0;
   S703_WELD_BUFF_DATA10.RBT9_BT_CODE_NO := W#16#0;
   S703_WELD_BUFF_DATA10.RBT9_WELD_COUNT := W#16#0;
   S703_WELD_BUFF_DATA10.RBT10_BT_CODE_NO := W#16#0;
   S703_WELD_BUFF_DATA10.RBT10_WELD_COUNT := W#16#0;
   S703_WELD_BUFF_DATA10.RBT11_BT_CODE_NO := W#16#0;
   S703_WELD_BUFF_DATA10.RBT11_WELD_COUNT := W#16#0;
   S703_WELD_BUFF_DATA10.RBT12_BT_CODE_NO := W#16#0;
   S703_WELD_BUFF_DATA10.RBT12_WELD_COUNT := W#16#0;
   S703_WELD_BUFF_DATA10.RBT13_BT_CODE_NO := W#16#0;
   S703_WELD_BUFF_DATA10.RBT13_WELD_COUNT := W#16#0;
   S703_WELD_BUFF_DATA10.RBT14_BT_CODE_NO := W#16#0;
   S703_WELD_BUFF_DATA10.RBT14_WELD_COUNT := W#16#0;
   S703_WELD_BUFF_DATA10.RBT15_BT_CODE_NO := W#16#0;
   S703_WELD_BUFF_DATA10.RBT15_WELD_COUNT := W#16#0;
   S703_WELD_BUFF_DATA10.RBT16_BT_CODE_NO := W#16#0;
   S703_WELD_BUFF_DATA10.RBT16_WELD_COUNT := W#16#0;
   S703_WELD_BUFF_DATA10.RBT17_BT_CODE_NO := W#16#0;
   S703_WELD_BUFF_DATA10.RBT17_WELD_COUNT := W#16#0;
   S703_WELD_BUFF_DATA10.RBT18_BT_CODE_NO := W#16#0;
   S703_WELD_BUFF_DATA10.RBT18_WELD_COUNT := W#16#0;
   S703_WELD_BUFF_DATA10.RBT19_BT_CODE_NO := W#16#0;
   S703_WELD_BUFF_DATA10.RBT19_WELD_COUNT := W#16#0;
   S703_WELD_BUFF_DATA10.RBT20_BT_CODE_NO := W#16#0;
   S703_WELD_BUFF_DATA10.RBT20_WELD_COUNT := W#16#0;
   S703_WELD_BUFF_DATA10.RBT21_BT_CODE_NO := W#16#0;
   S703_WELD_BUFF_DATA10.RBT21_WELD_COUNT := W#16#0;
   S703_WELD_BUFF_DATA10.RBT22_BT_CODE_NO := W#16#0;
   S703_WELD_BUFF_DATA10.RBT22_WELD_COUNT := W#16#0;
   S703_WELD_BUFF_DATA10.RBT23_BT_CODE_NO := W#16#0;
   S703_WELD_BUFF_DATA10.RBT23_WELD_COUNT := W#16#0;
   S703_WELD_BUFF_DATA10.RBT24_BT_CODE_NO := W#16#0;
   S703_WELD_BUFF_DATA10.RBT24_WELD_COUNT := W#16#0;
   S703_WELD_BUFF_DATA10.WELD_DETERMINES_RESULT := W#16#0;
   S703_WELD_BUFF_DATA10.WELD_CHECK_SUM := W#16#0;
   S703_WELD_BUFF_DATA10.SPARE1 := W#16#0;
   S704_WELD_BUFF_DATA1.STATION_MAIN := W#16#0;
   S704_WELD_BUFF_DATA1.DISTINCTION_LH_RH := W#16#0;
   S704_WELD_BUFF_DATA1.STAION_NUMBER := W#16#0;
   S704_WELD_BUFF_DATA1.VIN_NUMBER1 := W#16#0;
   S704_WELD_BUFF_DATA1.VIN_NUMBER2 := W#16#0;
   S704_WELD_BUFF_DATA1.VIN_NUMBER3 := W#16#0;
   S704_WELD_BUFF_DATA1.VIN_NUMBER4 := W#16#0;
   S704_WELD_BUFF_DATA1.SEQ_NUMBER1 := W#16#0;
   S704_WELD_BUFF_DATA1.SEQ_NUMBER2 := W#16#0;
   S704_WELD_BUFF_DATA1.RBT1_BT_CODE_NO := W#16#0;
   S704_WELD_BUFF_DATA1.RBT1_WELD_COUNT := W#16#0;
   S704_WELD_BUFF_DATA1.RBT2_BT_CODE_NO := W#16#0;
   S704_WELD_BUFF_DATA1.RBT2_WELD_COUNT := W#16#0;
   S704_WELD_BUFF_DATA1.RBT3_BT_CODE_NO := W#16#0;
   S704_WELD_BUFF_DATA1.RBT3_WELD_COUNT := W#16#0;
   S704_WELD_BUFF_DATA1.RBT4_BT_CODE_NO := W#16#0;
   S704_WELD_BUFF_DATA1.RBT4_WELD_COUNT := W#16#0;
   S704_WELD_BUFF_DATA1.RBT5_BT_CODE_NO := W#16#0;
   S704_WELD_BUFF_DATA1.RBT5_WELD_COUNT := W#16#0;
   S704_WELD_BUFF_DATA1.RBT6_BT_CODE_NO := W#16#0;
   S704_WELD_BUFF_DATA1.RBT6_WELD_COUNT := W#16#0;
   S704_WELD_BUFF_DATA1.RBT7_BT_CODE_NO := W#16#0;
   S704_WELD_BUFF_DATA1.RBT7_WELD_COUNT := W#16#0;
   S704_WELD_BUFF_DATA1.RBT8_BT_CODE_NO := W#16#0;
   S704_WELD_BUFF_DATA1.RBT8_WELD_COUNT := W#16#0;
   S704_WELD_BUFF_DATA1.RBT9_BT_CODE_NO := W#16#0;
   S704_WELD_BUFF_DATA1.RBT9_WELD_COUNT := W#16#0;
   S704_WELD_BUFF_DATA1.RBT10_BT_CODE_NO := W#16#0;
   S704_WELD_BUFF_DATA1.RBT10_WELD_COUNT := W#16#0;
   S704_WELD_BUFF_DATA1.RBT11_BT_CODE_NO := W#16#0;
   S704_WELD_BUFF_DATA1.RBT11_WELD_COUNT := W#16#0;
   S704_WELD_BUFF_DATA1.RBT12_BT_CODE_NO := W#16#0;
   S704_WELD_BUFF_DATA1.RBT12_WELD_COUNT := W#16#0;
   S704_WELD_BUFF_DATA1.RBT13_BT_CODE_NO := W#16#0;
   S704_WELD_BUFF_DATA1.RBT13_WELD_COUNT := W#16#0;
   S704_WELD_BUFF_DATA1.RBT14_BT_CODE_NO := W#16#0;
   S704_WELD_BUFF_DATA1.RBT14_WELD_COUNT := W#16#0;
   S704_WELD_BUFF_DATA1.RBT15_BT_CODE_NO := W#16#0;
   S704_WELD_BUFF_DATA1.RBT15_WELD_COUNT := W#16#0;
   S704_WELD_BUFF_DATA1.RBT16_BT_CODE_NO := W#16#0;
   S704_WELD_BUFF_DATA1.RBT16_WELD_COUNT := W#16#0;
   S704_WELD_BUFF_DATA1.RBT17_BT_CODE_NO := W#16#0;
   S704_WELD_BUFF_DATA1.RBT17_WELD_COUNT := W#16#0;
   S704_WELD_BUFF_DATA1.RBT18_BT_CODE_NO := W#16#0;
   S704_WELD_BUFF_DATA1.RBT18_WELD_COUNT := W#16#0;
   S704_WELD_BUFF_DATA1.RBT19_BT_CODE_NO := W#16#0;
   S704_WELD_BUFF_DATA1.RBT19_WELD_COUNT := W#16#0;
   S704_WELD_BUFF_DATA1.RBT20_BT_CODE_NO := W#16#0;
   S704_WELD_BUFF_DATA1.RBT20_WELD_COUNT := W#16#0;
   S704_WELD_BUFF_DATA1.RBT21_BT_CODE_NO := W#16#0;
   S704_WELD_BUFF_DATA1.RBT21_WELD_COUNT := W#16#0;
   S704_WELD_BUFF_DATA1.RBT22_BT_CODE_NO := W#16#0;
   S704_WELD_BUFF_DATA1.RBT22_WELD_COUNT := W#16#0;
   S704_WELD_BUFF_DATA1.RBT23_BT_CODE_NO := W#16#0;
   S704_WELD_BUFF_DATA1.RBT23_WELD_COUNT := W#16#0;
   S704_WELD_BUFF_DATA1.RBT24_BT_CODE_NO := W#16#0;
   S704_WELD_BUFF_DATA1.RBT24_WELD_COUNT := W#16#0;
   S704_WELD_BUFF_DATA1.WELD_DETERMINES_RESULT := W#16#0;
   S704_WELD_BUFF_DATA1.WELD_CHECK_SUM := W#16#0;
   S704_WELD_BUFF_DATA1.SPARE1 := W#16#0;
   S704_WELD_BUFF_DATA2.STATION_MAIN := W#16#0;
   S704_WELD_BUFF_DATA2.DISTINCTION_LH_RH := W#16#0;
   S704_WELD_BUFF_DATA2.STAION_NUMBER := W#16#0;
   S704_WELD_BUFF_DATA2.VIN_NUMBER1 := W#16#0;
   S704_WELD_BUFF_DATA2.VIN_NUMBER2 := W#16#0;
   S704_WELD_BUFF_DATA2.VIN_NUMBER3 := W#16#0;
   S704_WELD_BUFF_DATA2.VIN_NUMBER4 := W#16#0;
   S704_WELD_BUFF_DATA2.SEQ_NUMBER1 := W#16#0;
   S704_WELD_BUFF_DATA2.SEQ_NUMBER2 := W#16#0;
   S704_WELD_BUFF_DATA2.RBT1_BT_CODE_NO := W#16#0;
   S704_WELD_BUFF_DATA2.RBT1_WELD_COUNT := W#16#0;
   S704_WELD_BUFF_DATA2.RBT2_BT_CODE_NO := W#16#0;
   S704_WELD_BUFF_DATA2.RBT2_WELD_COUNT := W#16#0;
   S704_WELD_BUFF_DATA2.RBT3_BT_CODE_NO := W#16#0;
   S704_WELD_BUFF_DATA2.RBT3_WELD_COUNT := W#16#0;
   S704_WELD_BUFF_DATA2.RBT4_BT_CODE_NO := W#16#0;
   S704_WELD_BUFF_DATA2.RBT4_WELD_COUNT := W#16#0;
   S704_WELD_BUFF_DATA2.RBT5_BT_CODE_NO := W#16#0;
   S704_WELD_BUFF_DATA2.RBT5_WELD_COUNT := W#16#0;
   S704_WELD_BUFF_DATA2.RBT6_BT_CODE_NO := W#16#0;
   S704_WELD_BUFF_DATA2.RBT6_WELD_COUNT := W#16#0;
   S704_WELD_BUFF_DATA2.RBT7_BT_CODE_NO := W#16#0;
   S704_WELD_BUFF_DATA2.RBT7_WELD_COUNT := W#16#0;
   S704_WELD_BUFF_DATA2.RBT8_BT_CODE_NO := W#16#0;
   S704_WELD_BUFF_DATA2.RBT8_WELD_COUNT := W#16#0;
   S704_WELD_BUFF_DATA2.RBT9_BT_CODE_NO := W#16#0;
   S704_WELD_BUFF_DATA2.RBT9_WELD_COUNT := W#16#0;
   S704_WELD_BUFF_DATA2.RBT10_BT_CODE_NO := W#16#0;
   S704_WELD_BUFF_DATA2.RBT10_WELD_COUNT := W#16#0;
   S704_WELD_BUFF_DATA2.RBT11_BT_CODE_NO := W#16#0;
   S704_WELD_BUFF_DATA2.RBT11_WELD_COUNT := W#16#0;
   S704_WELD_BUFF_DATA2.RBT12_BT_CODE_NO := W#16#0;
   S704_WELD_BUFF_DATA2.RBT12_WELD_COUNT := W#16#0;
   S704_WELD_BUFF_DATA2.RBT13_BT_CODE_NO := W#16#0;
   S704_WELD_BUFF_DATA2.RBT13_WELD_COUNT := W#16#0;
   S704_WELD_BUFF_DATA2.RBT14_BT_CODE_NO := W#16#0;
   S704_WELD_BUFF_DATA2.RBT14_WELD_COUNT := W#16#0;
   S704_WELD_BUFF_DATA2.RBT15_BT_CODE_NO := W#16#0;
   S704_WELD_BUFF_DATA2.RBT15_WELD_COUNT := W#16#0;
   S704_WELD_BUFF_DATA2.RBT16_BT_CODE_NO := W#16#0;
   S704_WELD_BUFF_DATA2.RBT16_WELD_COUNT := W#16#0;
   S704_WELD_BUFF_DATA2.RBT17_BT_CODE_NO := W#16#0;
   S704_WELD_BUFF_DATA2.RBT17_WELD_COUNT := W#16#0;
   S704_WELD_BUFF_DATA2.RBT18_BT_CODE_NO := W#16#0;
   S704_WELD_BUFF_DATA2.RBT18_WELD_COUNT := W#16#0;
   S704_WELD_BUFF_DATA2.RBT19_BT_CODE_NO := W#16#0;
   S704_WELD_BUFF_DATA2.RBT19_WELD_COUNT := W#16#0;
   S704_WELD_BUFF_DATA2.RBT20_BT_CODE_NO := W#16#0;
   S704_WELD_BUFF_DATA2.RBT20_WELD_COUNT := W#16#0;
   S704_WELD_BUFF_DATA2.RBT21_BT_CODE_NO := W#16#0;
   S704_WELD_BUFF_DATA2.RBT21_WELD_COUNT := W#16#0;
   S704_WELD_BUFF_DATA2.RBT22_BT_CODE_NO := W#16#0;
   S704_WELD_BUFF_DATA2.RBT22_WELD_COUNT := W#16#0;
   S704_WELD_BUFF_DATA2.RBT23_BT_CODE_NO := W#16#0;
   S704_WELD_BUFF_DATA2.RBT23_WELD_COUNT := W#16#0;
   S704_WELD_BUFF_DATA2.RBT24_BT_CODE_NO := W#16#0;
   S704_WELD_BUFF_DATA2.RBT24_WELD_COUNT := W#16#0;
   S704_WELD_BUFF_DATA2.WELD_DETERMINES_RESULT := W#16#0;
   S704_WELD_BUFF_DATA2.WELD_CHECK_SUM := W#16#0;
   S704_WELD_BUFF_DATA2.SPARE1 := W#16#0;
   S704_WELD_BUFF_DATA3.STATION_MAIN := W#16#0;
   S704_WELD_BUFF_DATA3.DISTINCTION_LH_RH := W#16#0;
   S704_WELD_BUFF_DATA3.STAION_NUMBER := W#16#0;
   S704_WELD_BUFF_DATA3.VIN_NUMBER1 := W#16#0;
   S704_WELD_BUFF_DATA3.VIN_NUMBER2 := W#16#0;
   S704_WELD_BUFF_DATA3.VIN_NUMBER3 := W#16#0;
   S704_WELD_BUFF_DATA3.VIN_NUMBER4 := W#16#0;
   S704_WELD_BUFF_DATA3.SEQ_NUMBER1 := W#16#0;
   S704_WELD_BUFF_DATA3.SEQ_NUMBER2 := W#16#0;
   S704_WELD_BUFF_DATA3.RBT1_BT_CODE_NO := W#16#0;
   S704_WELD_BUFF_DATA3.RBT1_WELD_COUNT := W#16#0;
   S704_WELD_BUFF_DATA3.RBT2_BT_CODE_NO := W#16#0;
   S704_WELD_BUFF_DATA3.RBT2_WELD_COUNT := W#16#0;
   S704_WELD_BUFF_DATA3.RBT3_BT_CODE_NO := W#16#0;
   S704_WELD_BUFF_DATA3.RBT3_WELD_COUNT := W#16#0;
   S704_WELD_BUFF_DATA3.RBT4_BT_CODE_NO := W#16#0;
   S704_WELD_BUFF_DATA3.RBT4_WELD_COUNT := W#16#0;
   S704_WELD_BUFF_DATA3.RBT5_BT_CODE_NO := W#16#0;
   S704_WELD_BUFF_DATA3.RBT5_WELD_COUNT := W#16#0;
   S704_WELD_BUFF_DATA3.RBT6_BT_CODE_NO := W#16#0;
   S704_WELD_BUFF_DATA3.RBT6_WELD_COUNT := W#16#0;
   S704_WELD_BUFF_DATA3.RBT7_BT_CODE_NO := W#16#0;
   S704_WELD_BUFF_DATA3.RBT7_WELD_COUNT := W#16#0;
   S704_WELD_BUFF_DATA3.RBT8_BT_CODE_NO := W#16#0;
   S704_WELD_BUFF_DATA3.RBT8_WELD_COUNT := W#16#0;
   S704_WELD_BUFF_DATA3.RBT9_BT_CODE_NO := W#16#0;
   S704_WELD_BUFF_DATA3.RBT9_WELD_COUNT := W#16#0;
   S704_WELD_BUFF_DATA3.RBT10_BT_CODE_NO := W#16#0;
   S704_WELD_BUFF_DATA3.RBT10_WELD_COUNT := W#16#0;
   S704_WELD_BUFF_DATA3.RBT11_BT_CODE_NO := W#16#0;
   S704_WELD_BUFF_DATA3.RBT11_WELD_COUNT := W#16#0;
   S704_WELD_BUFF_DATA3.RBT12_BT_CODE_NO := W#16#0;
   S704_WELD_BUFF_DATA3.RBT12_WELD_COUNT := W#16#0;
   S704_WELD_BUFF_DATA3.RBT13_BT_CODE_NO := W#16#0;
   S704_WELD_BUFF_DATA3.RBT13_WELD_COUNT := W#16#0;
   S704_WELD_BUFF_DATA3.RBT14_BT_CODE_NO := W#16#0;
   S704_WELD_BUFF_DATA3.RBT14_WELD_COUNT := W#16#0;
   S704_WELD_BUFF_DATA3.RBT15_BT_CODE_NO := W#16#0;
   S704_WELD_BUFF_DATA3.RBT15_WELD_COUNT := W#16#0;
   S704_WELD_BUFF_DATA3.RBT16_BT_CODE_NO := W#16#0;
   S704_WELD_BUFF_DATA3.RBT16_WELD_COUNT := W#16#0;
   S704_WELD_BUFF_DATA3.RBT17_BT_CODE_NO := W#16#0;
   S704_WELD_BUFF_DATA3.RBT17_WELD_COUNT := W#16#0;
   S704_WELD_BUFF_DATA3.RBT18_BT_CODE_NO := W#16#0;
   S704_WELD_BUFF_DATA3.RBT18_WELD_COUNT := W#16#0;
   S704_WELD_BUFF_DATA3.RBT19_BT_CODE_NO := W#16#0;
   S704_WELD_BUFF_DATA3.RBT19_WELD_COUNT := W#16#0;
   S704_WELD_BUFF_DATA3.RBT20_BT_CODE_NO := W#16#0;
   S704_WELD_BUFF_DATA3.RBT20_WELD_COUNT := W#16#0;
   S704_WELD_BUFF_DATA3.RBT21_BT_CODE_NO := W#16#0;
   S704_WELD_BUFF_DATA3.RBT21_WELD_COUNT := W#16#0;
   S704_WELD_BUFF_DATA3.RBT22_BT_CODE_NO := W#16#0;
   S704_WELD_BUFF_DATA3.RBT22_WELD_COUNT := W#16#0;
   S704_WELD_BUFF_DATA3.RBT23_BT_CODE_NO := W#16#0;
   S704_WELD_BUFF_DATA3.RBT23_WELD_COUNT := W#16#0;
   S704_WELD_BUFF_DATA3.RBT24_BT_CODE_NO := W#16#0;
   S704_WELD_BUFF_DATA3.RBT24_WELD_COUNT := W#16#0;
   S704_WELD_BUFF_DATA3.WELD_DETERMINES_RESULT := W#16#0;
   S704_WELD_BUFF_DATA3.WELD_CHECK_SUM := W#16#0;
   S704_WELD_BUFF_DATA3.SPARE1 := W#16#0;
   S704_WELD_BUFF_DATA4.STATION_MAIN := W#16#0;
   S704_WELD_BUFF_DATA4.DISTINCTION_LH_RH := W#16#0;
   S704_WELD_BUFF_DATA4.STAION_NUMBER := W#16#0;
   S704_WELD_BUFF_DATA4.VIN_NUMBER1 := W#16#0;
   S704_WELD_BUFF_DATA4.VIN_NUMBER2 := W#16#0;
   S704_WELD_BUFF_DATA4.VIN_NUMBER3 := W#16#0;
   S704_WELD_BUFF_DATA4.VIN_NUMBER4 := W#16#0;
   S704_WELD_BUFF_DATA4.SEQ_NUMBER1 := W#16#0;
   S704_WELD_BUFF_DATA4.SEQ_NUMBER2 := W#16#0;
   S704_WELD_BUFF_DATA4.RBT1_BT_CODE_NO := W#16#0;
   S704_WELD_BUFF_DATA4.RBT1_WELD_COUNT := W#16#0;
   S704_WELD_BUFF_DATA4.RBT2_BT_CODE_NO := W#16#0;
   S704_WELD_BUFF_DATA4.RBT2_WELD_COUNT := W#16#0;
   S704_WELD_BUFF_DATA4.RBT3_BT_CODE_NO := W#16#0;
   S704_WELD_BUFF_DATA4.RBT3_WELD_COUNT := W#16#0;
   S704_WELD_BUFF_DATA4.RBT4_BT_CODE_NO := W#16#0;
   S704_WELD_BUFF_DATA4.RBT4_WELD_COUNT := W#16#0;
   S704_WELD_BUFF_DATA4.RBT5_BT_CODE_NO := W#16#0;
   S704_WELD_BUFF_DATA4.RBT5_WELD_COUNT := W#16#0;
   S704_WELD_BUFF_DATA4.RBT6_BT_CODE_NO := W#16#0;
   S704_WELD_BUFF_DATA4.RBT6_WELD_COUNT := W#16#0;
   S704_WELD_BUFF_DATA4.RBT7_BT_CODE_NO := W#16#0;
   S704_WELD_BUFF_DATA4.RBT7_WELD_COUNT := W#16#0;
   S704_WELD_BUFF_DATA4.RBT8_BT_CODE_NO := W#16#0;
   S704_WELD_BUFF_DATA4.RBT8_WELD_COUNT := W#16#0;
   S704_WELD_BUFF_DATA4.RBT9_BT_CODE_NO := W#16#0;
   S704_WELD_BUFF_DATA4.RBT9_WELD_COUNT := W#16#0;
   S704_WELD_BUFF_DATA4.RBT10_BT_CODE_NO := W#16#0;
   S704_WELD_BUFF_DATA4.RBT10_WELD_COUNT := W#16#0;
   S704_WELD_BUFF_DATA4.RBT11_BT_CODE_NO := W#16#0;
   S704_WELD_BUFF_DATA4.RBT11_WELD_COUNT := W#16#0;
   S704_WELD_BUFF_DATA4.RBT12_BT_CODE_NO := W#16#0;
   S704_WELD_BUFF_DATA4.RBT12_WELD_COUNT := W#16#0;
   S704_WELD_BUFF_DATA4.RBT13_BT_CODE_NO := W#16#0;
   S704_WELD_BUFF_DATA4.RBT13_WELD_COUNT := W#16#0;
   S704_WELD_BUFF_DATA4.RBT14_BT_CODE_NO := W#16#0;
   S704_WELD_BUFF_DATA4.RBT14_WELD_COUNT := W#16#0;
   S704_WELD_BUFF_DATA4.RBT15_BT_CODE_NO := W#16#0;
   S704_WELD_BUFF_DATA4.RBT15_WELD_COUNT := W#16#0;
   S704_WELD_BUFF_DATA4.RBT16_BT_CODE_NO := W#16#0;
   S704_WELD_BUFF_DATA4.RBT16_WELD_COUNT := W#16#0;
   S704_WELD_BUFF_DATA4.RBT17_BT_CODE_NO := W#16#0;
   S704_WELD_BUFF_DATA4.RBT17_WELD_COUNT := W#16#0;
   S704_WELD_BUFF_DATA4.RBT18_BT_CODE_NO := W#16#0;
   S704_WELD_BUFF_DATA4.RBT18_WELD_COUNT := W#16#0;
   S704_WELD_BUFF_DATA4.RBT19_BT_CODE_NO := W#16#0;
   S704_WELD_BUFF_DATA4.RBT19_WELD_COUNT := W#16#0;
   S704_WELD_BUFF_DATA4.RBT20_BT_CODE_NO := W#16#0;
   S704_WELD_BUFF_DATA4.RBT20_WELD_COUNT := W#16#0;
   S704_WELD_BUFF_DATA4.RBT21_BT_CODE_NO := W#16#0;
   S704_WELD_BUFF_DATA4.RBT21_WELD_COUNT := W#16#0;
   S704_WELD_BUFF_DATA4.RBT22_BT_CODE_NO := W#16#0;
   S704_WELD_BUFF_DATA4.RBT22_WELD_COUNT := W#16#0;
   S704_WELD_BUFF_DATA4.RBT23_BT_CODE_NO := W#16#0;
   S704_WELD_BUFF_DATA4.RBT23_WELD_COUNT := W#16#0;
   S704_WELD_BUFF_DATA4.RBT24_BT_CODE_NO := W#16#0;
   S704_WELD_BUFF_DATA4.RBT24_WELD_COUNT := W#16#0;
   S704_WELD_BUFF_DATA4.WELD_DETERMINES_RESULT := W#16#0;
   S704_WELD_BUFF_DATA4.WELD_CHECK_SUM := W#16#0;
   S704_WELD_BUFF_DATA4.SPARE1 := W#16#0;
   S704_WELD_BUFF_DATA5.STATION_MAIN := W#16#0;
   S704_WELD_BUFF_DATA5.DISTINCTION_LH_RH := W#16#0;
   S704_WELD_BUFF_DATA5.STAION_NUMBER := W#16#0;
   S704_WELD_BUFF_DATA5.VIN_NUMBER1 := W#16#0;
   S704_WELD_BUFF_DATA5.VIN_NUMBER2 := W#16#0;
   S704_WELD_BUFF_DATA5.VIN_NUMBER3 := W#16#0;
   S704_WELD_BUFF_DATA5.VIN_NUMBER4 := W#16#0;
   S704_WELD_BUFF_DATA5.SEQ_NUMBER1 := W#16#0;
   S704_WELD_BUFF_DATA5.SEQ_NUMBER2 := W#16#0;
   S704_WELD_BUFF_DATA5.RBT1_BT_CODE_NO := W#16#0;
   S704_WELD_BUFF_DATA5.RBT1_WELD_COUNT := W#16#0;
   S704_WELD_BUFF_DATA5.RBT2_BT_CODE_NO := W#16#0;
   S704_WELD_BUFF_DATA5.RBT2_WELD_COUNT := W#16#0;
   S704_WELD_BUFF_DATA5.RBT3_BT_CODE_NO := W#16#0;
   S704_WELD_BUFF_DATA5.RBT3_WELD_COUNT := W#16#0;
   S704_WELD_BUFF_DATA5.RBT4_BT_CODE_NO := W#16#0;
   S704_WELD_BUFF_DATA5.RBT4_WELD_COUNT := W#16#0;
   S704_WELD_BUFF_DATA5.RBT5_BT_CODE_NO := W#16#0;
   S704_WELD_BUFF_DATA5.RBT5_WELD_COUNT := W#16#0;
   S704_WELD_BUFF_DATA5.RBT6_BT_CODE_NO := W#16#0;
   S704_WELD_BUFF_DATA5.RBT6_WELD_COUNT := W#16#0;
   S704_WELD_BUFF_DATA5.RBT7_BT_CODE_NO := W#16#0;
   S704_WELD_BUFF_DATA5.RBT7_WELD_COUNT := W#16#0;
   S704_WELD_BUFF_DATA5.RBT8_BT_CODE_NO := W#16#0;
   S704_WELD_BUFF_DATA5.RBT8_WELD_COUNT := W#16#0;
   S704_WELD_BUFF_DATA5.RBT9_BT_CODE_NO := W#16#0;
   S704_WELD_BUFF_DATA5.RBT9_WELD_COUNT := W#16#0;
   S704_WELD_BUFF_DATA5.RBT10_BT_CODE_NO := W#16#0;
   S704_WELD_BUFF_DATA5.RBT10_WELD_COUNT := W#16#0;
   S704_WELD_BUFF_DATA5.RBT11_BT_CODE_NO := W#16#0;
   S704_WELD_BUFF_DATA5.RBT11_WELD_COUNT := W#16#0;
   S704_WELD_BUFF_DATA5.RBT12_BT_CODE_NO := W#16#0;
   S704_WELD_BUFF_DATA5.RBT12_WELD_COUNT := W#16#0;
   S704_WELD_BUFF_DATA5.RBT13_BT_CODE_NO := W#16#0;
   S704_WELD_BUFF_DATA5.RBT13_WELD_COUNT := W#16#0;
   S704_WELD_BUFF_DATA5.RBT14_BT_CODE_NO := W#16#0;
   S704_WELD_BUFF_DATA5.RBT14_WELD_COUNT := W#16#0;
   S704_WELD_BUFF_DATA5.RBT15_BT_CODE_NO := W#16#0;
   S704_WELD_BUFF_DATA5.RBT15_WELD_COUNT := W#16#0;
   S704_WELD_BUFF_DATA5.RBT16_BT_CODE_NO := W#16#0;
   S704_WELD_BUFF_DATA5.RBT16_WELD_COUNT := W#16#0;
   S704_WELD_BUFF_DATA5.RBT17_BT_CODE_NO := W#16#0;
   S704_WELD_BUFF_DATA5.RBT17_WELD_COUNT := W#16#0;
   S704_WELD_BUFF_DATA5.RBT18_BT_CODE_NO := W#16#0;
   S704_WELD_BUFF_DATA5.RBT18_WELD_COUNT := W#16#0;
   S704_WELD_BUFF_DATA5.RBT19_BT_CODE_NO := W#16#0;
   S704_WELD_BUFF_DATA5.RBT19_WELD_COUNT := W#16#0;
   S704_WELD_BUFF_DATA5.RBT20_BT_CODE_NO := W#16#0;
   S704_WELD_BUFF_DATA5.RBT20_WELD_COUNT := W#16#0;
   S704_WELD_BUFF_DATA5.RBT21_BT_CODE_NO := W#16#0;
   S704_WELD_BUFF_DATA5.RBT21_WELD_COUNT := W#16#0;
   S704_WELD_BUFF_DATA5.RBT22_BT_CODE_NO := W#16#0;
   S704_WELD_BUFF_DATA5.RBT22_WELD_COUNT := W#16#0;
   S704_WELD_BUFF_DATA5.RBT23_BT_CODE_NO := W#16#0;
   S704_WELD_BUFF_DATA5.RBT23_WELD_COUNT := W#16#0;
   S704_WELD_BUFF_DATA5.RBT24_BT_CODE_NO := W#16#0;
   S704_WELD_BUFF_DATA5.RBT24_WELD_COUNT := W#16#0;
   S704_WELD_BUFF_DATA5.WELD_DETERMINES_RESULT := W#16#0;
   S704_WELD_BUFF_DATA5.WELD_CHECK_SUM := W#16#0;
   S704_WELD_BUFF_DATA5.SPARE1 := W#16#0;
   S704_WELD_BUFF_DATA6.STATION_MAIN := W#16#0;
   S704_WELD_BUFF_DATA6.DISTINCTION_LH_RH := W#16#0;
   S704_WELD_BUFF_DATA6.STAION_NUMBER := W#16#0;
   S704_WELD_BUFF_DATA6.VIN_NUMBER1 := W#16#0;
   S704_WELD_BUFF_DATA6.VIN_NUMBER2 := W#16#0;
   S704_WELD_BUFF_DATA6.VIN_NUMBER3 := W#16#0;
   S704_WELD_BUFF_DATA6.VIN_NUMBER4 := W#16#0;
   S704_WELD_BUFF_DATA6.SEQ_NUMBER1 := W#16#0;
   S704_WELD_BUFF_DATA6.SEQ_NUMBER2 := W#16#0;
   S704_WELD_BUFF_DATA6.RBT1_BT_CODE_NO := W#16#0;
   S704_WELD_BUFF_DATA6.RBT1_WELD_COUNT := W#16#0;
   S704_WELD_BUFF_DATA6.RBT2_BT_CODE_NO := W#16#0;
   S704_WELD_BUFF_DATA6.RBT2_WELD_COUNT := W#16#0;
   S704_WELD_BUFF_DATA6.RBT3_BT_CODE_NO := W#16#0;
   S704_WELD_BUFF_DATA6.RBT3_WELD_COUNT := W#16#0;
   S704_WELD_BUFF_DATA6.RBT4_BT_CODE_NO := W#16#0;
   S704_WELD_BUFF_DATA6.RBT4_WELD_COUNT := W#16#0;
   S704_WELD_BUFF_DATA6.RBT5_BT_CODE_NO := W#16#0;
   S704_WELD_BUFF_DATA6.RBT5_WELD_COUNT := W#16#0;
   S704_WELD_BUFF_DATA6.RBT6_BT_CODE_NO := W#16#0;
   S704_WELD_BUFF_DATA6.RBT6_WELD_COUNT := W#16#0;
   S704_WELD_BUFF_DATA6.RBT7_BT_CODE_NO := W#16#0;
   S704_WELD_BUFF_DATA6.RBT7_WELD_COUNT := W#16#0;
   S704_WELD_BUFF_DATA6.RBT8_BT_CODE_NO := W#16#0;
   S704_WELD_BUFF_DATA6.RBT8_WELD_COUNT := W#16#0;
   S704_WELD_BUFF_DATA6.RBT9_BT_CODE_NO := W#16#0;
   S704_WELD_BUFF_DATA6.RBT9_WELD_COUNT := W#16#0;
   S704_WELD_BUFF_DATA6.RBT10_BT_CODE_NO := W#16#0;
   S704_WELD_BUFF_DATA6.RBT10_WELD_COUNT := W#16#0;
   S704_WELD_BUFF_DATA6.RBT11_BT_CODE_NO := W#16#0;
   S704_WELD_BUFF_DATA6.RBT11_WELD_COUNT := W#16#0;
   S704_WELD_BUFF_DATA6.RBT12_BT_CODE_NO := W#16#0;
   S704_WELD_BUFF_DATA6.RBT12_WELD_COUNT := W#16#0;
   S704_WELD_BUFF_DATA6.RBT13_BT_CODE_NO := W#16#0;
   S704_WELD_BUFF_DATA6.RBT13_WELD_COUNT := W#16#0;
   S704_WELD_BUFF_DATA6.RBT14_BT_CODE_NO := W#16#0;
   S704_WELD_BUFF_DATA6.RBT14_WELD_COUNT := W#16#0;
   S704_WELD_BUFF_DATA6.RBT15_BT_CODE_NO := W#16#0;
   S704_WELD_BUFF_DATA6.RBT15_WELD_COUNT := W#16#0;
   S704_WELD_BUFF_DATA6.RBT16_BT_CODE_NO := W#16#0;
   S704_WELD_BUFF_DATA6.RBT16_WELD_COUNT := W#16#0;
   S704_WELD_BUFF_DATA6.RBT17_BT_CODE_NO := W#16#0;
   S704_WELD_BUFF_DATA6.RBT17_WELD_COUNT := W#16#0;
   S704_WELD_BUFF_DATA6.RBT18_BT_CODE_NO := W#16#0;
   S704_WELD_BUFF_DATA6.RBT18_WELD_COUNT := W#16#0;
   S704_WELD_BUFF_DATA6.RBT19_BT_CODE_NO := W#16#0;
   S704_WELD_BUFF_DATA6.RBT19_WELD_COUNT := W#16#0;
   S704_WELD_BUFF_DATA6.RBT20_BT_CODE_NO := W#16#0;
   S704_WELD_BUFF_DATA6.RBT20_WELD_COUNT := W#16#0;
   S704_WELD_BUFF_DATA6.RBT21_BT_CODE_NO := W#16#0;
   S704_WELD_BUFF_DATA6.RBT21_WELD_COUNT := W#16#0;
   S704_WELD_BUFF_DATA6.RBT22_BT_CODE_NO := W#16#0;
   S704_WELD_BUFF_DATA6.RBT22_WELD_COUNT := W#16#0;
   S704_WELD_BUFF_DATA6.RBT23_BT_CODE_NO := W#16#0;
   S704_WELD_BUFF_DATA6.RBT23_WELD_COUNT := W#16#0;
   S704_WELD_BUFF_DATA6.RBT24_BT_CODE_NO := W#16#0;
   S704_WELD_BUFF_DATA6.RBT24_WELD_COUNT := W#16#0;
   S704_WELD_BUFF_DATA6.WELD_DETERMINES_RESULT := W#16#0;
   S704_WELD_BUFF_DATA6.WELD_CHECK_SUM := W#16#0;
   S704_WELD_BUFF_DATA6.SPARE1 := W#16#0;
   S704_WELD_BUFF_DATA7.STATION_MAIN := W#16#0;
   S704_WELD_BUFF_DATA7.DISTINCTION_LH_RH := W#16#0;
   S704_WELD_BUFF_DATA7.STAION_NUMBER := W#16#0;
   S704_WELD_BUFF_DATA7.VIN_NUMBER1 := W#16#0;
   S704_WELD_BUFF_DATA7.VIN_NUMBER2 := W#16#0;
   S704_WELD_BUFF_DATA7.VIN_NUMBER3 := W#16#0;
   S704_WELD_BUFF_DATA7.VIN_NUMBER4 := W#16#0;
   S704_WELD_BUFF_DATA7.SEQ_NUMBER1 := W#16#0;
   S704_WELD_BUFF_DATA7.SEQ_NUMBER2 := W#16#0;
   S704_WELD_BUFF_DATA7.RBT1_BT_CODE_NO := W#16#0;
   S704_WELD_BUFF_DATA7.RBT1_WELD_COUNT := W#16#0;
   S704_WELD_BUFF_DATA7.RBT2_BT_CODE_NO := W#16#0;
   S704_WELD_BUFF_DATA7.RBT2_WELD_COUNT := W#16#0;
   S704_WELD_BUFF_DATA7.RBT3_BT_CODE_NO := W#16#0;
   S704_WELD_BUFF_DATA7.RBT3_WELD_COUNT := W#16#0;
   S704_WELD_BUFF_DATA7.RBT4_BT_CODE_NO := W#16#0;
   S704_WELD_BUFF_DATA7.RBT4_WELD_COUNT := W#16#0;
   S704_WELD_BUFF_DATA7.RBT5_BT_CODE_NO := W#16#0;
   S704_WELD_BUFF_DATA7.RBT5_WELD_COUNT := W#16#0;
   S704_WELD_BUFF_DATA7.RBT6_BT_CODE_NO := W#16#0;
   S704_WELD_BUFF_DATA7.RBT6_WELD_COUNT := W#16#0;
   S704_WELD_BUFF_DATA7.RBT7_BT_CODE_NO := W#16#0;
   S704_WELD_BUFF_DATA7.RBT7_WELD_COUNT := W#16#0;
   S704_WELD_BUFF_DATA7.RBT8_BT_CODE_NO := W#16#0;
   S704_WELD_BUFF_DATA7.RBT8_WELD_COUNT := W#16#0;
   S704_WELD_BUFF_DATA7.RBT9_BT_CODE_NO := W#16#0;
   S704_WELD_BUFF_DATA7.RBT9_WELD_COUNT := W#16#0;
   S704_WELD_BUFF_DATA7.RBT10_BT_CODE_NO := W#16#0;
   S704_WELD_BUFF_DATA7.RBT10_WELD_COUNT := W#16#0;
   S704_WELD_BUFF_DATA7.RBT11_BT_CODE_NO := W#16#0;
   S704_WELD_BUFF_DATA7.RBT11_WELD_COUNT := W#16#0;
   S704_WELD_BUFF_DATA7.RBT12_BT_CODE_NO := W#16#0;
   S704_WELD_BUFF_DATA7.RBT12_WELD_COUNT := W#16#0;
   S704_WELD_BUFF_DATA7.RBT13_BT_CODE_NO := W#16#0;
   S704_WELD_BUFF_DATA7.RBT13_WELD_COUNT := W#16#0;
   S704_WELD_BUFF_DATA7.RBT14_BT_CODE_NO := W#16#0;
   S704_WELD_BUFF_DATA7.RBT14_WELD_COUNT := W#16#0;
   S704_WELD_BUFF_DATA7.RBT15_BT_CODE_NO := W#16#0;
   S704_WELD_BUFF_DATA7.RBT15_WELD_COUNT := W#16#0;
   S704_WELD_BUFF_DATA7.RBT16_BT_CODE_NO := W#16#0;
   S704_WELD_BUFF_DATA7.RBT16_WELD_COUNT := W#16#0;
   S704_WELD_BUFF_DATA7.RBT17_BT_CODE_NO := W#16#0;
   S704_WELD_BUFF_DATA7.RBT17_WELD_COUNT := W#16#0;
   S704_WELD_BUFF_DATA7.RBT18_BT_CODE_NO := W#16#0;
   S704_WELD_BUFF_DATA7.RBT18_WELD_COUNT := W#16#0;
   S704_WELD_BUFF_DATA7.RBT19_BT_CODE_NO := W#16#0;
   S704_WELD_BUFF_DATA7.RBT19_WELD_COUNT := W#16#0;
   S704_WELD_BUFF_DATA7.RBT20_BT_CODE_NO := W#16#0;
   S704_WELD_BUFF_DATA7.RBT20_WELD_COUNT := W#16#0;
   S704_WELD_BUFF_DATA7.RBT21_BT_CODE_NO := W#16#0;
   S704_WELD_BUFF_DATA7.RBT21_WELD_COUNT := W#16#0;
   S704_WELD_BUFF_DATA7.RBT22_BT_CODE_NO := W#16#0;
   S704_WELD_BUFF_DATA7.RBT22_WELD_COUNT := W#16#0;
   S704_WELD_BUFF_DATA7.RBT23_BT_CODE_NO := W#16#0;
   S704_WELD_BUFF_DATA7.RBT23_WELD_COUNT := W#16#0;
   S704_WELD_BUFF_DATA7.RBT24_BT_CODE_NO := W#16#0;
   S704_WELD_BUFF_DATA7.RBT24_WELD_COUNT := W#16#0;
   S704_WELD_BUFF_DATA7.WELD_DETERMINES_RESULT := W#16#0;
   S704_WELD_BUFF_DATA7.WELD_CHECK_SUM := W#16#0;
   S704_WELD_BUFF_DATA7.SPARE1 := W#16#0;
   S704_WELD_BUFF_DATA8.STATION_MAIN := W#16#0;
   S704_WELD_BUFF_DATA8.DISTINCTION_LH_RH := W#16#0;
   S704_WELD_BUFF_DATA8.STAION_NUMBER := W#16#0;
   S704_WELD_BUFF_DATA8.VIN_NUMBER1 := W#16#0;
   S704_WELD_BUFF_DATA8.VIN_NUMBER2 := W#16#0;
   S704_WELD_BUFF_DATA8.VIN_NUMBER3 := W#16#0;
   S704_WELD_BUFF_DATA8.VIN_NUMBER4 := W#16#0;
   S704_WELD_BUFF_DATA8.SEQ_NUMBER1 := W#16#0;
   S704_WELD_BUFF_DATA8.SEQ_NUMBER2 := W#16#0;
   S704_WELD_BUFF_DATA8.RBT1_BT_CODE_NO := W#16#0;
   S704_WELD_BUFF_DATA8.RBT1_WELD_COUNT := W#16#0;
   S704_WELD_BUFF_DATA8.RBT2_BT_CODE_NO := W#16#0;
   S704_WELD_BUFF_DATA8.RBT2_WELD_COUNT := W#16#0;
   S704_WELD_BUFF_DATA8.RBT3_BT_CODE_NO := W#16#0;
   S704_WELD_BUFF_DATA8.RBT3_WELD_COUNT := W#16#0;
   S704_WELD_BUFF_DATA8.RBT4_BT_CODE_NO := W#16#0;
   S704_WELD_BUFF_DATA8.RBT4_WELD_COUNT := W#16#0;
   S704_WELD_BUFF_DATA8.RBT5_BT_CODE_NO := W#16#0;
   S704_WELD_BUFF_DATA8.RBT5_WELD_COUNT := W#16#0;
   S704_WELD_BUFF_DATA8.RBT6_BT_CODE_NO := W#16#0;
   S704_WELD_BUFF_DATA8.RBT6_WELD_COUNT := W#16#0;
   S704_WELD_BUFF_DATA8.RBT7_BT_CODE_NO := W#16#0;
   S704_WELD_BUFF_DATA8.RBT7_WELD_COUNT := W#16#0;
   S704_WELD_BUFF_DATA8.RBT8_BT_CODE_NO := W#16#0;
   S704_WELD_BUFF_DATA8.RBT8_WELD_COUNT := W#16#0;
   S704_WELD_BUFF_DATA8.RBT9_BT_CODE_NO := W#16#0;
   S704_WELD_BUFF_DATA8.RBT9_WELD_COUNT := W#16#0;
   S704_WELD_BUFF_DATA8.RBT10_BT_CODE_NO := W#16#0;
   S704_WELD_BUFF_DATA8.RBT10_WELD_COUNT := W#16#0;
   S704_WELD_BUFF_DATA8.RBT11_BT_CODE_NO := W#16#0;
   S704_WELD_BUFF_DATA8.RBT11_WELD_COUNT := W#16#0;
   S704_WELD_BUFF_DATA8.RBT12_BT_CODE_NO := W#16#0;
   S704_WELD_BUFF_DATA8.RBT12_WELD_COUNT := W#16#0;
   S704_WELD_BUFF_DATA8.RBT13_BT_CODE_NO := W#16#0;
   S704_WELD_BUFF_DATA8.RBT13_WELD_COUNT := W#16#0;
   S704_WELD_BUFF_DATA8.RBT14_BT_CODE_NO := W#16#0;
   S704_WELD_BUFF_DATA8.RBT14_WELD_COUNT := W#16#0;
   S704_WELD_BUFF_DATA8.RBT15_BT_CODE_NO := W#16#0;
   S704_WELD_BUFF_DATA8.RBT15_WELD_COUNT := W#16#0;
   S704_WELD_BUFF_DATA8.RBT16_BT_CODE_NO := W#16#0;
   S704_WELD_BUFF_DATA8.RBT16_WELD_COUNT := W#16#0;
   S704_WELD_BUFF_DATA8.RBT17_BT_CODE_NO := W#16#0;
   S704_WELD_BUFF_DATA8.RBT17_WELD_COUNT := W#16#0;
   S704_WELD_BUFF_DATA8.RBT18_BT_CODE_NO := W#16#0;
   S704_WELD_BUFF_DATA8.RBT18_WELD_COUNT := W#16#0;
   S704_WELD_BUFF_DATA8.RBT19_BT_CODE_NO := W#16#0;
   S704_WELD_BUFF_DATA8.RBT19_WELD_COUNT := W#16#0;
   S704_WELD_BUFF_DATA8.RBT20_BT_CODE_NO := W#16#0;
   S704_WELD_BUFF_DATA8.RBT20_WELD_COUNT := W#16#0;
   S704_WELD_BUFF_DATA8.RBT21_BT_CODE_NO := W#16#0;
   S704_WELD_BUFF_DATA8.RBT21_WELD_COUNT := W#16#0;
   S704_WELD_BUFF_DATA8.RBT22_BT_CODE_NO := W#16#0;
   S704_WELD_BUFF_DATA8.RBT22_WELD_COUNT := W#16#0;
   S704_WELD_BUFF_DATA8.RBT23_BT_CODE_NO := W#16#0;
   S704_WELD_BUFF_DATA8.RBT23_WELD_COUNT := W#16#0;
   S704_WELD_BUFF_DATA8.RBT24_BT_CODE_NO := W#16#0;
   S704_WELD_BUFF_DATA8.RBT24_WELD_COUNT := W#16#0;
   S704_WELD_BUFF_DATA8.WELD_DETERMINES_RESULT := W#16#0;
   S704_WELD_BUFF_DATA8.WELD_CHECK_SUM := W#16#0;
   S704_WELD_BUFF_DATA8.SPARE1 := W#16#0;
   S704_WELD_BUFF_DATA9.STATION_MAIN := W#16#0;
   S704_WELD_BUFF_DATA9.DISTINCTION_LH_RH := W#16#0;
   S704_WELD_BUFF_DATA9.STAION_NUMBER := W#16#0;
   S704_WELD_BUFF_DATA9.VIN_NUMBER1 := W#16#0;
   S704_WELD_BUFF_DATA9.VIN_NUMBER2 := W#16#0;
   S704_WELD_BUFF_DATA9.VIN_NUMBER3 := W#16#0;
   S704_WELD_BUFF_DATA9.VIN_NUMBER4 := W#16#0;
   S704_WELD_BUFF_DATA9.SEQ_NUMBER1 := W#16#0;
   S704_WELD_BUFF_DATA9.SEQ_NUMBER2 := W#16#0;
   S704_WELD_BUFF_DATA9.RBT1_BT_CODE_NO := W#16#0;
   S704_WELD_BUFF_DATA9.RBT1_WELD_COUNT := W#16#0;
   S704_WELD_BUFF_DATA9.RBT2_BT_CODE_NO := W#16#0;
   S704_WELD_BUFF_DATA9.RBT2_WELD_COUNT := W#16#0;
   S704_WELD_BUFF_DATA9.RBT3_BT_CODE_NO := W#16#0;
   S704_WELD_BUFF_DATA9.RBT3_WELD_COUNT := W#16#0;
   S704_WELD_BUFF_DATA9.RBT4_BT_CODE_NO := W#16#0;
   S704_WELD_BUFF_DATA9.RBT4_WELD_COUNT := W#16#0;
   S704_WELD_BUFF_DATA9.RBT5_BT_CODE_NO := W#16#0;
   S704_WELD_BUFF_DATA9.RBT5_WELD_COUNT := W#16#0;
   S704_WELD_BUFF_DATA9.RBT6_BT_CODE_NO := W#16#0;
   S704_WELD_BUFF_DATA9.RBT6_WELD_COUNT := W#16#0;
   S704_WELD_BUFF_DATA9.RBT7_BT_CODE_NO := W#16#0;
   S704_WELD_BUFF_DATA9.RBT7_WELD_COUNT := W#16#0;
   S704_WELD_BUFF_DATA9.RBT8_BT_CODE_NO := W#16#0;
   S704_WELD_BUFF_DATA9.RBT8_WELD_COUNT := W#16#0;
   S704_WELD_BUFF_DATA9.RBT9_BT_CODE_NO := W#16#0;
   S704_WELD_BUFF_DATA9.RBT9_WELD_COUNT := W#16#0;
   S704_WELD_BUFF_DATA9.RBT10_BT_CODE_NO := W#16#0;
   S704_WELD_BUFF_DATA9.RBT10_WELD_COUNT := W#16#0;
   S704_WELD_BUFF_DATA9.RBT11_BT_CODE_NO := W#16#0;
   S704_WELD_BUFF_DATA9.RBT11_WELD_COUNT := W#16#0;
   S704_WELD_BUFF_DATA9.RBT12_BT_CODE_NO := W#16#0;
   S704_WELD_BUFF_DATA9.RBT12_WELD_COUNT := W#16#0;
   S704_WELD_BUFF_DATA9.RBT13_BT_CODE_NO := W#16#0;
   S704_WELD_BUFF_DATA9.RBT13_WELD_COUNT := W#16#0;
   S704_WELD_BUFF_DATA9.RBT14_BT_CODE_NO := W#16#0;
   S704_WELD_BUFF_DATA9.RBT14_WELD_COUNT := W#16#0;
   S704_WELD_BUFF_DATA9.RBT15_BT_CODE_NO := W#16#0;
   S704_WELD_BUFF_DATA9.RBT15_WELD_COUNT := W#16#0;
   S704_WELD_BUFF_DATA9.RBT16_BT_CODE_NO := W#16#0;
   S704_WELD_BUFF_DATA9.RBT16_WELD_COUNT := W#16#0;
   S704_WELD_BUFF_DATA9.RBT17_BT_CODE_NO := W#16#0;
   S704_WELD_BUFF_DATA9.RBT17_WELD_COUNT := W#16#0;
   S704_WELD_BUFF_DATA9.RBT18_BT_CODE_NO := W#16#0;
   S704_WELD_BUFF_DATA9.RBT18_WELD_COUNT := W#16#0;
   S704_WELD_BUFF_DATA9.RBT19_BT_CODE_NO := W#16#0;
   S704_WELD_BUFF_DATA9.RBT19_WELD_COUNT := W#16#0;
   S704_WELD_BUFF_DATA9.RBT20_BT_CODE_NO := W#16#0;
   S704_WELD_BUFF_DATA9.RBT20_WELD_COUNT := W#16#0;
   S704_WELD_BUFF_DATA9.RBT21_BT_CODE_NO := W#16#0;
   S704_WELD_BUFF_DATA9.RBT21_WELD_COUNT := W#16#0;
   S704_WELD_BUFF_DATA9.RBT22_BT_CODE_NO := W#16#0;
   S704_WELD_BUFF_DATA9.RBT22_WELD_COUNT := W#16#0;
   S704_WELD_BUFF_DATA9.RBT23_BT_CODE_NO := W#16#0;
   S704_WELD_BUFF_DATA9.RBT23_WELD_COUNT := W#16#0;
   S704_WELD_BUFF_DATA9.RBT24_BT_CODE_NO := W#16#0;
   S704_WELD_BUFF_DATA9.RBT24_WELD_COUNT := W#16#0;
   S704_WELD_BUFF_DATA9.WELD_DETERMINES_RESULT := W#16#0;
   S704_WELD_BUFF_DATA9.WELD_CHECK_SUM := W#16#0;
   S704_WELD_BUFF_DATA9.SPARE1 := W#16#0;
   S704_WELD_BUFF_DATA10.STATION_MAIN := W#16#0;
   S704_WELD_BUFF_DATA10.DISTINCTION_LH_RH := W#16#0;
   S704_WELD_BUFF_DATA10.STAION_NUMBER := W#16#0;
   S704_WELD_BUFF_DATA10.VIN_NUMBER1 := W#16#0;
   S704_WELD_BUFF_DATA10.VIN_NUMBER2 := W#16#0;
   S704_WELD_BUFF_DATA10.VIN_NUMBER3 := W#16#0;
   S704_WELD_BUFF_DATA10.VIN_NUMBER4 := W#16#0;
   S704_WELD_BUFF_DATA10.SEQ_NUMBER1 := W#16#0;
   S704_WELD_BUFF_DATA10.SEQ_NUMBER2 := W#16#0;
   S704_WELD_BUFF_DATA10.RBT1_BT_CODE_NO := W#16#0;
   S704_WELD_BUFF_DATA10.RBT1_WELD_COUNT := W#16#0;
   S704_WELD_BUFF_DATA10.RBT2_BT_CODE_NO := W#16#0;
   S704_WELD_BUFF_DATA10.RBT2_WELD_COUNT := W#16#0;
   S704_WELD_BUFF_DATA10.RBT3_BT_CODE_NO := W#16#0;
   S704_WELD_BUFF_DATA10.RBT3_WELD_COUNT := W#16#0;
   S704_WELD_BUFF_DATA10.RBT4_BT_CODE_NO := W#16#0;
   S704_WELD_BUFF_DATA10.RBT4_WELD_COUNT := W#16#0;
   S704_WELD_BUFF_DATA10.RBT5_BT_CODE_NO := W#16#0;
   S704_WELD_BUFF_DATA10.RBT5_WELD_COUNT := W#16#0;
   S704_WELD_BUFF_DATA10.RBT6_BT_CODE_NO := W#16#0;
   S704_WELD_BUFF_DATA10.RBT6_WELD_COUNT := W#16#0;
   S704_WELD_BUFF_DATA10.RBT7_BT_CODE_NO := W#16#0;
   S704_WELD_BUFF_DATA10.RBT7_WELD_COUNT := W#16#0;
   S704_WELD_BUFF_DATA10.RBT8_BT_CODE_NO := W#16#0;
   S704_WELD_BUFF_DATA10.RBT8_WELD_COUNT := W#16#0;
   S704_WELD_BUFF_DATA10.RBT9_BT_CODE_NO := W#16#0;
   S704_WELD_BUFF_DATA10.RBT9_WELD_COUNT := W#16#0;
   S704_WELD_BUFF_DATA10.RBT10_BT_CODE_NO := W#16#0;
   S704_WELD_BUFF_DATA10.RBT10_WELD_COUNT := W#16#0;
   S704_WELD_BUFF_DATA10.RBT11_BT_CODE_NO := W#16#0;
   S704_WELD_BUFF_DATA10.RBT11_WELD_COUNT := W#16#0;
   S704_WELD_BUFF_DATA10.RBT12_BT_CODE_NO := W#16#0;
   S704_WELD_BUFF_DATA10.RBT12_WELD_COUNT := W#16#0;
   S704_WELD_BUFF_DATA10.RBT13_BT_CODE_NO := W#16#0;
   S704_WELD_BUFF_DATA10.RBT13_WELD_COUNT := W#16#0;
   S704_WELD_BUFF_DATA10.RBT14_BT_CODE_NO := W#16#0;
   S704_WELD_BUFF_DATA10.RBT14_WELD_COUNT := W#16#0;
   S704_WELD_BUFF_DATA10.RBT15_BT_CODE_NO := W#16#0;
   S704_WELD_BUFF_DATA10.RBT15_WELD_COUNT := W#16#0;
   S704_WELD_BUFF_DATA10.RBT16_BT_CODE_NO := W#16#0;
   S704_WELD_BUFF_DATA10.RBT16_WELD_COUNT := W#16#0;
   S704_WELD_BUFF_DATA10.RBT17_BT_CODE_NO := W#16#0;
   S704_WELD_BUFF_DATA10.RBT17_WELD_COUNT := W#16#0;
   S704_WELD_BUFF_DATA10.RBT18_BT_CODE_NO := W#16#0;
   S704_WELD_BUFF_DATA10.RBT18_WELD_COUNT := W#16#0;
   S704_WELD_BUFF_DATA10.RBT19_BT_CODE_NO := W#16#0;
   S704_WELD_BUFF_DATA10.RBT19_WELD_COUNT := W#16#0;
   S704_WELD_BUFF_DATA10.RBT20_BT_CODE_NO := W#16#0;
   S704_WELD_BUFF_DATA10.RBT20_WELD_COUNT := W#16#0;
   S704_WELD_BUFF_DATA10.RBT21_BT_CODE_NO := W#16#0;
   S704_WELD_BUFF_DATA10.RBT21_WELD_COUNT := W#16#0;
   S704_WELD_BUFF_DATA10.RBT22_BT_CODE_NO := W#16#0;
   S704_WELD_BUFF_DATA10.RBT22_WELD_COUNT := W#16#0;
   S704_WELD_BUFF_DATA10.RBT23_BT_CODE_NO := W#16#0;
   S704_WELD_BUFF_DATA10.RBT23_WELD_COUNT := W#16#0;
   S704_WELD_BUFF_DATA10.RBT24_BT_CODE_NO := W#16#0;
   S704_WELD_BUFF_DATA10.RBT24_WELD_COUNT := W#16#0;
   S704_WELD_BUFF_DATA10.WELD_DETERMINES_RESULT := W#16#0;
   S704_WELD_BUFF_DATA10.WELD_CHECK_SUM := W#16#0;
   S704_WELD_BUFF_DATA10.SPARE1 := W#16#0;
   S704_WELD_BUFF_DATA11.STATION_MAIN := W#16#0;
   S704_WELD_BUFF_DATA11.DISTINCTION_LH_RH := W#16#0;
   S704_WELD_BUFF_DATA11.STAION_NUMBER := W#16#0;
   S704_WELD_BUFF_DATA11.VIN_NUMBER1 := W#16#0;
   S704_WELD_BUFF_DATA11.VIN_NUMBER2 := W#16#0;
   S704_WELD_BUFF_DATA11.VIN_NUMBER3 := W#16#0;
   S704_WELD_BUFF_DATA11.VIN_NUMBER4 := W#16#0;
   S704_WELD_BUFF_DATA11.SEQ_NUMBER1 := W#16#0;
   S704_WELD_BUFF_DATA11.SEQ_NUMBER2 := W#16#0;
   S704_WELD_BUFF_DATA11.RBT1_BT_CODE_NO := W#16#0;
   S704_WELD_BUFF_DATA11.RBT1_WELD_COUNT := W#16#0;
   S704_WELD_BUFF_DATA11.RBT2_BT_CODE_NO := W#16#0;
   S704_WELD_BUFF_DATA11.RBT2_WELD_COUNT := W#16#0;
   S704_WELD_BUFF_DATA11.RBT3_BT_CODE_NO := W#16#0;
   S704_WELD_BUFF_DATA11.RBT3_WELD_COUNT := W#16#0;
   S704_WELD_BUFF_DATA11.RBT4_BT_CODE_NO := W#16#0;
   S704_WELD_BUFF_DATA11.RBT4_WELD_COUNT := W#16#0;
   S704_WELD_BUFF_DATA11.RBT5_BT_CODE_NO := W#16#0;
   S704_WELD_BUFF_DATA11.RBT5_WELD_COUNT := W#16#0;
   S704_WELD_BUFF_DATA11.RBT6_BT_CODE_NO := W#16#0;
   S704_WELD_BUFF_DATA11.RBT6_WELD_COUNT := W#16#0;
   S704_WELD_BUFF_DATA11.RBT7_BT_CODE_NO := W#16#0;
   S704_WELD_BUFF_DATA11.RBT7_WELD_COUNT := W#16#0;
   S704_WELD_BUFF_DATA11.RBT8_BT_CODE_NO := W#16#0;
   S704_WELD_BUFF_DATA11.RBT8_WELD_COUNT := W#16#0;
   S704_WELD_BUFF_DATA11.RBT9_BT_CODE_NO := W#16#0;
   S704_WELD_BUFF_DATA11.RBT9_WELD_COUNT := W#16#0;
   S704_WELD_BUFF_DATA11.RBT10_BT_CODE_NO := W#16#0;
   S704_WELD_BUFF_DATA11.RBT10_WELD_COUNT := W#16#0;
   S704_WELD_BUFF_DATA11.RBT11_BT_CODE_NO := W#16#0;
   S704_WELD_BUFF_DATA11.RBT11_WELD_COUNT := W#16#0;
   S704_WELD_BUFF_DATA11.RBT12_BT_CODE_NO := W#16#0;
   S704_WELD_BUFF_DATA11.RBT12_WELD_COUNT := W#16#0;
   S704_WELD_BUFF_DATA11.RBT13_BT_CODE_NO := W#16#0;
   S704_WELD_BUFF_DATA11.RBT13_WELD_COUNT := W#16#0;
   S704_WELD_BUFF_DATA11.RBT14_BT_CODE_NO := W#16#0;
   S704_WELD_BUFF_DATA11.RBT14_WELD_COUNT := W#16#0;
   S704_WELD_BUFF_DATA11.RBT15_BT_CODE_NO := W#16#0;
   S704_WELD_BUFF_DATA11.RBT15_WELD_COUNT := W#16#0;
   S704_WELD_BUFF_DATA11.RBT16_BT_CODE_NO := W#16#0;
   S704_WELD_BUFF_DATA11.RBT16_WELD_COUNT := W#16#0;
   S704_WELD_BUFF_DATA11.RBT17_BT_CODE_NO := W#16#0;
   S704_WELD_BUFF_DATA11.RBT17_WELD_COUNT := W#16#0;
   S704_WELD_BUFF_DATA11.RBT18_BT_CODE_NO := W#16#0;
   S704_WELD_BUFF_DATA11.RBT18_WELD_COUNT := W#16#0;
   S704_WELD_BUFF_DATA11.RBT19_BT_CODE_NO := W#16#0;
   S704_WELD_BUFF_DATA11.RBT19_WELD_COUNT := W#16#0;
   S704_WELD_BUFF_DATA11.RBT20_BT_CODE_NO := W#16#0;
   S704_WELD_BUFF_DATA11.RBT20_WELD_COUNT := W#16#0;
   S704_WELD_BUFF_DATA11.RBT21_BT_CODE_NO := W#16#0;
   S704_WELD_BUFF_DATA11.RBT21_WELD_COUNT := W#16#0;
   S704_WELD_BUFF_DATA11.RBT22_BT_CODE_NO := W#16#0;
   S704_WELD_BUFF_DATA11.RBT22_WELD_COUNT := W#16#0;
   S704_WELD_BUFF_DATA11.RBT23_BT_CODE_NO := W#16#0;
   S704_WELD_BUFF_DATA11.RBT23_WELD_COUNT := W#16#0;
   S704_WELD_BUFF_DATA11.RBT24_BT_CODE_NO := W#16#0;
   S704_WELD_BUFF_DATA11.RBT24_WELD_COUNT := W#16#0;
   S704_WELD_BUFF_DATA11.WELD_DETERMINES_RESULT := W#16#0;
   S704_WELD_BUFF_DATA11.WELD_CHECK_SUM := W#16#0;
   S704_WELD_BUFF_DATA11.SPARE1 := W#16#0;
   S704_WELD_BUFF_DATA21.STATION_MAIN := W#16#0;
   S704_WELD_BUFF_DATA21.DISTINCTION_LH_RH := W#16#0;
   S704_WELD_BUFF_DATA21.STAION_NUMBER := W#16#0;
   S704_WELD_BUFF_DATA21.VIN_NUMBER1 := W#16#0;
   S704_WELD_BUFF_DATA21.VIN_NUMBER2 := W#16#0;
   S704_WELD_BUFF_DATA21.VIN_NUMBER3 := W#16#0;
   S704_WELD_BUFF_DATA21.VIN_NUMBER4 := W#16#0;
   S704_WELD_BUFF_DATA21.SEQ_NUMBER1 := W#16#0;
   S704_WELD_BUFF_DATA21.SEQ_NUMBER2 := W#16#0;
   S704_WELD_BUFF_DATA21.RBT1_BT_CODE_NO := W#16#0;
   S704_WELD_BUFF_DATA21.RBT1_WELD_COUNT := W#16#0;
   S704_WELD_BUFF_DATA21.RBT2_BT_CODE_NO := W#16#0;
   S704_WELD_BUFF_DATA21.RBT2_WELD_COUNT := W#16#0;
   S704_WELD_BUFF_DATA21.RBT3_BT_CODE_NO := W#16#0;
   S704_WELD_BUFF_DATA21.RBT3_WELD_COUNT := W#16#0;
   S704_WELD_BUFF_DATA21.RBT4_BT_CODE_NO := W#16#0;
   S704_WELD_BUFF_DATA21.RBT4_WELD_COUNT := W#16#0;
   S704_WELD_BUFF_DATA21.RBT5_BT_CODE_NO := W#16#0;
   S704_WELD_BUFF_DATA21.RBT5_WELD_COUNT := W#16#0;
   S704_WELD_BUFF_DATA21.RBT6_BT_CODE_NO := W#16#0;
   S704_WELD_BUFF_DATA21.RBT6_WELD_COUNT := W#16#0;
   S704_WELD_BUFF_DATA21.RBT7_BT_CODE_NO := W#16#0;
   S704_WELD_BUFF_DATA21.RBT7_WELD_COUNT := W#16#0;
   S704_WELD_BUFF_DATA21.RBT8_BT_CODE_NO := W#16#0;
   S704_WELD_BUFF_DATA21.RBT8_WELD_COUNT := W#16#0;
   S704_WELD_BUFF_DATA21.RBT9_BT_CODE_NO := W#16#0;
   S704_WELD_BUFF_DATA21.RBT9_WELD_COUNT := W#16#0;
   S704_WELD_BUFF_DATA21.RBT10_BT_CODE_NO := W#16#0;
   S704_WELD_BUFF_DATA21.RBT10_WELD_COUNT := W#16#0;
   S704_WELD_BUFF_DATA21.RBT11_BT_CODE_NO := W#16#0;
   S704_WELD_BUFF_DATA21.RBT11_WELD_COUNT := W#16#0;
   S704_WELD_BUFF_DATA21.RBT12_BT_CODE_NO := W#16#0;
   S704_WELD_BUFF_DATA21.RBT12_WELD_COUNT := W#16#0;
   S704_WELD_BUFF_DATA21.RBT13_BT_CODE_NO := W#16#0;
   S704_WELD_BUFF_DATA21.RBT13_WELD_COUNT := W#16#0;
   S704_WELD_BUFF_DATA21.RBT14_BT_CODE_NO := W#16#0;
   S704_WELD_BUFF_DATA21.RBT14_WELD_COUNT := W#16#0;
   S704_WELD_BUFF_DATA21.RBT15_BT_CODE_NO := W#16#0;
   S704_WELD_BUFF_DATA21.RBT15_WELD_COUNT := W#16#0;
   S704_WELD_BUFF_DATA21.RBT16_BT_CODE_NO := W#16#0;
   S704_WELD_BUFF_DATA21.RBT16_WELD_COUNT := W#16#0;
   S704_WELD_BUFF_DATA21.RBT17_BT_CODE_NO := W#16#0;
   S704_WELD_BUFF_DATA21.RBT17_WELD_COUNT := W#16#0;
   S704_WELD_BUFF_DATA21.RBT18_BT_CODE_NO := W#16#0;
   S704_WELD_BUFF_DATA21.RBT18_WELD_COUNT := W#16#0;
   S704_WELD_BUFF_DATA21.RBT19_BT_CODE_NO := W#16#0;
   S704_WELD_BUFF_DATA21.RBT19_WELD_COUNT := W#16#0;
   S704_WELD_BUFF_DATA21.RBT20_BT_CODE_NO := W#16#0;
   S704_WELD_BUFF_DATA21.RBT20_WELD_COUNT := W#16#0;
   S704_WELD_BUFF_DATA21.RBT21_BT_CODE_NO := W#16#0;
   S704_WELD_BUFF_DATA21.RBT21_WELD_COUNT := W#16#0;
   S704_WELD_BUFF_DATA21.RBT22_BT_CODE_NO := W#16#0;
   S704_WELD_BUFF_DATA21.RBT22_WELD_COUNT := W#16#0;
   S704_WELD_BUFF_DATA21.RBT23_BT_CODE_NO := W#16#0;
   S704_WELD_BUFF_DATA21.RBT23_WELD_COUNT := W#16#0;
   S704_WELD_BUFF_DATA21.RBT24_BT_CODE_NO := W#16#0;
   S704_WELD_BUFF_DATA21.RBT24_WELD_COUNT := W#16#0;
   S704_WELD_BUFF_DATA21.WELD_DETERMINES_RESULT := W#16#0;
   S704_WELD_BUFF_DATA21.WELD_CHECK_SUM := W#16#0;
   S704_WELD_BUFF_DATA21.SPARE1 := W#16#0;
   S704_WELD_BUFF_DATA31.STATION_MAIN := W#16#0;
   S704_WELD_BUFF_DATA31.DISTINCTION_LH_RH := W#16#0;
   S704_WELD_BUFF_DATA31.STAION_NUMBER := W#16#0;
   S704_WELD_BUFF_DATA31.VIN_NUMBER1 := W#16#0;
   S704_WELD_BUFF_DATA31.VIN_NUMBER2 := W#16#0;
   S704_WELD_BUFF_DATA31.VIN_NUMBER3 := W#16#0;
   S704_WELD_BUFF_DATA31.VIN_NUMBER4 := W#16#0;
   S704_WELD_BUFF_DATA31.SEQ_NUMBER1 := W#16#0;
   S704_WELD_BUFF_DATA31.SEQ_NUMBER2 := W#16#0;
   S704_WELD_BUFF_DATA31.RBT1_BT_CODE_NO := W#16#0;
   S704_WELD_BUFF_DATA31.RBT1_WELD_COUNT := W#16#0;
